LIN {X 0,Y 151.915,Z 503.399,A -85,B 0,C 180,E1 -24424.924,E2 -24424.924} C_VEL
LIN {X 0,Y 153.961,Z 512.067,A -85,B 0,C 180,E1 -24426.981,E2 -24426.981} C_VEL
LIN {X 0,Y 155.485,Z 521.164,A -85,B 0,C 180,E1 -24429.257,E2 -24429.257} C_VEL
LIN {X 0,Y 152.235,Z 533.845,A -85,B 0,C 180,E1 -24432.383,E2 -24432.383} C_VEL
LIN {X 0,Y 149.159,Z 545.494,A -85,B 0,C 180,E1 -24435.973,E2 -24435.973} C_VEL
LIN {X 0,Y 146.128,Z 556.818,A -85,B 0,C 180,E1 -24440.309,E2 -24440.309} C_VEL
LIN {X 0,Y 143.834,Z 566.337,A -85,B 0,C 180,E1 -24444.838,E2 -24444.838} C_VEL
LIN {X 0,Y 142.226,Z 574.336,A -85,B 0,C 180,E1 -24449.568,E2 -24449.568} C_VEL
LIN {X 0,Y 141.026,Z 581.744,A -85,B 0,C 180,E1 -24455.034,E2 -24455.034} C_VEL
LIN {X 0,Y 140.53,Z 587.875,A -85,B 0,C 180,E1 -24460.838,E2 -24460.838} C_VEL
LIN {X 0,Y 140.751,Z 591.758,A -85,B 0,C 180,E1 -24465.542,E2 -24465.542} C_VEL
LIN {X 0,Y 142.113,Z 595.406,A -85,B 0,C 180,E1 -24471.514,E2 -24471.514} C_VEL
LIN {X 0,Y 144.598,Z 597.709,A -85,B 0,C 180,E1 -24477.214,E2 -24477.214} C_VEL
LIN {X 0,Y 148.347,Z 598.825,A -85,B 0,C 180,E1 -24482.715,E2 -24482.715} C_VEL
LIN {X 0,Y 153.36,Z 598.771,A -85,B 0,C 180,E1 -24487.902,E2 -24487.902} C_VEL
LIN {X 0,Y 159.682,Z 597.562,A -85,B 0,C 180,E1 -24492.712,E2 -24492.712} C_VEL
LIN {X 0,Y 167.08,Z 595.209,A -85,B 0,C 180,E1 -24497.124,E2 -24497.124} C_VEL
LIN {X 0,Y 175.627,Z 591.631,A -85,B 0,C 180,E1 -24501.109,E2 -24501.109} C_VEL
LIN {X 0,Y 185.071,Z 586.803,A -85,B 0,C 180,E1 -24504.69,E2 -24504.69} C_VEL
LIN {X 0,Y 195.365,Z 580.517,A -85,B 0,C 180,E1 -24507.882,E2 -24507.882} C_VEL
LIN {X 0,Y 198.021,Z 578.731,A -85,B 0,C 180,E1 -24508.628,E2 -24508.628} C_VEL
LIN {X 0,Y 199.744,Z 577.522,A -85,B 0,C 180,E1 -24509.511,E2 -24509.511} C_VEL
LIN {X 0,Y 200.149,Z 577.047,A -85,B 0,C 180,E1 -24511.783,E2 -24511.783} C_VEL
LIN {X 0,Y 199.933,Z 577.424,A -85,B 0,C 180,E1 -24514.224,E2 -24514.224} C_VEL
LIN {X 0,Y 199.181,Z 578.642,A -85,B 0,C 180,E1 -24516.858,E2 -24516.858} C_VEL
LIN {X 0,Y 198.163,Z 580.069,A -85,B 0,C 180,E1 -24518.718,E2 -24518.718} C_VEL
LIN {X 0,Y 194.723,Z 583.259,A -85,B 0,C 180,E1 -24520.719,E2 -24520.719} C_VEL
LIN {X 0,Y 192.674,Z 584.987,A -85,B 0,C 180,E1 -24521.604,E2 -24521.604} C_VEL
LIN {X 0,Y 182.603,Z 591.982,A -85,B 0,C 180,E1 -24524.601,E2 -24524.601} C_VEL
LIN {X 0,Y 175.435,Z 596.39,A -85,B 0,C 180,E1 -24527.077,E2 -24527.077} C_VEL
LIN {X 0,Y 169.007,Z 600.188,A -85,B 0,C 180,E1 -24529.869,E2 -24529.869} C_VEL
LIN {X 0,Y 159.468,Z 605.111,A -85,B 0,C 180,E1 -24535.046,E2 -24535.046} C_VEL
LIN {X 0,Y 153.08,Z 607.936,A -85,B 0,C 180,E1 -24539.668,E2 -24539.668} C_VEL
LIN {X 0,Y 147.919,Z 609.705,A -85,B 0,C 180,E1 -24544.684,E2 -24544.684} C_VEL
LIN {X 0,Y 144.261,Z 610.461,A -85,B 0,C 180,E1 -24550.061,E2 -24550.061} C_VEL
LIN {X 0,Y 141.949,Z 610.176,A -85,B 0,C 180,E1 -24555.667,E2 -24555.667} C_VEL
LIN {X 0,Y 141.165,Z 608.842,A -85,B 0,C 180,E1 -24561.411,E2 -24561.411} C_VEL
LIN {X 0,Y 141.409,Z 606.295,A -85,B 0,C 180,E1 -24567.151,E2 -24567.151} C_VEL
LIN {X 0,Y 141.696,Z 604.494,A -85,B 0,C 180,E1 -24570,E2 -24570} C_VEL
LIN {X 0,Y 141.625,Z 600.931,A -85,B 0,C 180,E1 -24574.269,E2 -24574.269} C_VEL
LIN {X 0,Y 141.705,Z 596.358,A -85,B 0,C 180,E1 -24578.557,E2 -24578.557} C_VEL
LIN {X 0,Y 142.445,Z 589.643,A -85,B 0,C 180,E1 -24583.553,E2 -24583.553} C_VEL
LIN {X 0,Y 143.855,Z 581.253,A -85,B 0,C 180,E1 -24588.515,E2 -24588.515} C_VEL
LIN {X 0,Y 146.252,Z 571.401,A -85,B 0,C 180,E1 -24593.174,E2 -24593.174} C_VEL
LIN {X 0,Y 149.185,Z 560.252,A -85,B 0,C 180,E1 -24597.342,E2 -24597.342} C_VEL
LIN {X 0,Y 151.473,Z 551.924,A -85,B 0,C 180,E1 -24599.918,E2 -24599.918} C_VEL
LIN {X 0,Y 151.337,Z 542.468,A -85,B 0,C 180,E1 -24602.552,E2 -24602.552} C_VEL
LIN {X 0,Y 150.687,Z 529.752,A -85,B 0,C 180,E1 -24605.661,E2 -24605.661} C_VEL
LIN {X 0,Y 149.785,Z 516.716,A -85,B 0,C 180,E1 -24608.385,E2 -24608.385} C_VEL
LIN {X 0,Y 148.397,Z 501.688,A -85,B 0,C 180,E1 -24611.025,E2 -24611.025} C_VEL
LIN {X 0,Y 148.196,Z 499.899,A -85,B 0,C 180,E1 -24611.307,E2 -24611.307} C_VEL
LIN {X 0,Y 147.031,Z 496.512,A -85,B 0,C 180,E1 -24611.96,E2 -24611.96} C_VEL
LIN {X 0,Y 144.85,Z 493.641,A -85,B 0,C 180,E1 -24612.684,E2 -24612.684} C_VEL
LIN {X 0,Y 139.14,Z 487.285,A -85,B 0,C 180,E1 -24614.413,E2 -24614.413} C_VEL
LIN {X 0,Y 137.741,Z 483.867,A -85,B 0,C 180,E1 -24615.056,E2 -24615.056} C_VEL
LIN {X 0,Y 137.534,Z 482.616,A -85,B 0,C 180,E1 -24615.344,E2 -24615.344} C_VEL
LIN {X 0,Y 136.786,Z 479.643,A -85,B 0,C 180,E1 -24620.415,E2 -24620.415} C_VEL
LIN {X 0,Y 136.409,Z 477.116,A -85,B 0,C 180,E1 -24625.029,E2 -24625.029} C_VEL
LIN {X 0,Y 136.147,Z 477.149,A -85,B 0,C 180,E1 -24632.317,E2 -24632.317} C_VEL
LIN {X 0,Y 136.243,Z 477.139,A -85,B 0,C 180,E1 -24638.833,E2 -24638.833} C_VEL
LIN {X 0,Y 136.285,Z 477.129,A -85,B 0,C 180,E1 -24645.059,E2 -24645.059} C_VEL
LIN {X 0,Y 136.495,Z 477.107,A -85,B 0,C 180,E1 -24648.115,E2 -24648.115} C_VEL
LIN {X 0,Y 136.59,Z 477.092,A -85,B 0,C 180,E1 -24651.121,E2 -24651.121} C_VEL
LIN {X 0,Y 137.132,Z 477.026,A -85,B 0,C 180,E1 -24660.001,E2 -24660.001} C_VEL
LIN {X 0,Y 136.59,Z 477.092,A -85,B 0,C 180,E1 -24668.88,E2 -24668.88} C_VEL
LIN {X 0,Y 136.49,Z 477.103,A -85,B 0,C 180,E1 -24671.955,E2 -24671.955} C_VEL
LIN {X 0,Y 136.243,Z 477.136,A -85,B 0,C 180,E1 -24678.03,E2 -24678.03} C_VEL
LIN {X 0,Y 136.197,Z 477.142,A -85,B 0,C 180,E1 -24681.749,E2 -24681.749} C_VEL
LIN {X 0,Y 136.1,Z 477.151,A -85,B 0,C 180,E1 -24688.617,E2 -24688.617} C_VEL
LIN {X 0,Y 136.079,Z 477.157,A -85,B 0,C 180,E1 -24694.62,E2 -24694.62} C_VEL
LIN {X 0,Y 136.051,Z 477.16,A -85,B 0,C 180,E1 -24699.209,E2 -24699.209} C_VEL
LIN {X 0,Y 136.004,Z 477.168,A -85,B 0,C 180,E1 -24703.661,E2 -24703.661} C_VEL
LIN {X 0,Y 136.036,Z 477.162,A -85,B 0,C 180,E1 -24707.809,E2 -24707.809} C_VEL
LIN {X 0,Y 136.058,Z 477.162,A -85,B 0,C 180,E1 -24711.695,E2 -24711.695} C_VEL
LIN {X 0,Y 136.092,Z 477.152,A -85,B 0,C 180,E1 -24715.718,E2 -24715.718} C_VEL
LIN {X 0,Y 136.149,Z 477.145,A -85,B 0,C 180,E1 -24722.317,E2 -24722.317} C_VEL
LIN {X 0,Y 136.246,Z 477.138,A -85,B 0,C 180,E1 -24728.834,E2 -24728.834} C_VEL
LIN {X 0,Y 136.271,Z 477.134,A -85,B 0,C 180,E1 -24735.057,E2 -24735.057} C_VEL
LIN {X 0,Y 136.434,Z 477.113,A -85,B 0,C 180,E1 -24738.165,E2 -24738.165} C_VEL
LIN {X 0,Y 136.552,Z 477.094,A -85,B 0,C 180,E1 -24741.118,E2 -24741.118} C_VEL
LIN {X 0,Y 137.136,Z 477.021,A -85,B 0,C 180,E1 -24750,E2 -24750} C_VEL
LIN {X 0,Y 136.556,Z 477.091,A -85,B 0,C 180,E1 -24758.882,E2 -24758.882} C_VEL
LIN {X 0,Y 136.443,Z 477.113,A -85,B 0,C 180,E1 -24761.89,E2 -24761.89} C_VEL
LIN {X 0,Y 136.249,Z 477.134,A -85,B 0,C 180,E1 -24768.028,E2 -24768.028} C_VEL
LIN {X 0,Y 136.201,Z 477.144,A -85,B 0,C 180,E1 -24771.749,E2 -24771.749} C_VEL
LIN {X 0,Y 136.166,Z 477.215,A -85,B 0,C 180,E1 -24778.003,E2 -24778.003} C_VEL
LIN {X 0,Y 137.968,Z 482.338,A -85,B 0,C 180,E1 -24779.083,E2 -24779.083} C_VEL
LIN {X 0,Y 142.002,Z 494.173,A -85,B 0,C 180,E1 -24781.725,E2 -24781.725} C_VEL
LIN {X 0,Y 145.517,Z 506.485,A -85,B 0,C 180,E1 -24784.659,E2 -24784.659} C_VEL
LIN {X 0,Y 147.515,Z 515.552,A -85,B 0,C 180,E1 -24786.976,E2 -24786.976} C_VEL
LIN {X 0,Y 148.445,Z 520.908,A -85,B 0,C 180,E1 -24788.417,E2 -24788.417} C_VEL
LIN {X 0,Y 147.335,Z 526.449,A -85,B 0,C 180,E1 -24789.772,E2 -24789.772} C_VEL
LIN {X 0,Y 143.953,Z 538.976,A -85,B 0,C 180,E1 -24793.272,E2 -24793.272} C_VEL
LIN {X 0,Y 140.81,Z 550.38,A -85,B 0,C 180,E1 -24797.298,E2 -24797.298} C_VEL
LIN {X 0,Y 138.22,Z 559.95,A -85,B 0,C 180,E1 -24801.473,E2 -24801.473} C_VEL
LIN {X 0,Y 136.13,Z 569.001,A -85,B 0,C 180,E1 -24806.319,E2 -24806.319} C_VEL
LIN {X 0,Y 134.673,Z 576.356,A -85,B 0,C 180,E1 -24811.136,E2 -24811.136} C_VEL
LIN {X 0,Y 133.697,Z 583.307,A -85,B 0,C 180,E1 -24816.78,E2 -24816.78} C_VEL
LIN {X 0,Y 133.467,Z 588.029,A -85,B 0,C 180,E1 -24821.582,E2 -24821.582} C_VEL
LIN {X 0,Y 134.029,Z 592.858,A -85,B 0,C 180,E1 -24827.892,E2 -24827.892} C_VEL
LIN {X 0,Y 135.854,Z 596.28,A -85,B 0,C 180,E1 -24834.061,E2 -24834.061} C_VEL
LIN {X 0,Y 138.982,Z 598.438,A -85,B 0,C 180,E1 -24839.999,E2 -24839.999} C_VEL
LIN {X 0,Y 143.394,Z 599.427,A -85,B 0,C 180,E1 -24845.625,E2 -24845.625} C_VEL
LIN {X 0,Y 149.209,Z 599.265,A -85,B 0,C 180,E1 -24850.859,E2 -24850.859} C_VEL
LIN {X 0,Y 156.236,Z 597.981,A -85,B 0,C 180,E1 -24855.658,E2 -24855.658} C_VEL
LIN {X 0,Y 164.656,Z 595.448,A -85,B 0,C 180,E1 -24860.115,E2 -24860.115} C_VEL
LIN {X 0,Y 173.636,Z 591.918,A -85,B 0,C 180,E1 -24863.875,E2 -24863.875} C_VEL
LIN {X 0,Y 183.769,Z 586.966,A -85,B 0,C 180,E1 -24867.317,E2 -24867.317} C_VEL
LIN {X 0,Y 191.889,Z 582.364,A -85,B 0,C 180,E1 -24869.633,E2 -24869.633} C_VEL
LIN {X 0,Y 193.883,Z 581.13,A -85,B 0,C 180,E1 -24870.496,E2 -24870.496} C_VEL
LIN {X 0,Y 194.153,Z 581.028,A -85,B 0,C 180,E1 -24872.886,E2 -24872.886} C_VEL
LIN {X 0,Y 193.576,Z 581.831,A -85,B 0,C 180,E1 -24875.513,E2 -24875.513} C_VEL
LIN {X 0,Y 193.043,Z 582.549,A -85,B 0,C 180,E1 -24876.781,E2 -24876.781} C_VEL
LIN {X 0,Y 191.011,Z 584.458,A -85,B 0,C 180,E1 -24878.718,E2 -24878.718} C_VEL
LIN {X 0,Y 188.142,Z 586.678,A -85,B 0,C 180,E1 -24880.025,E2 -24880.025} C_VEL
LIN {X 0,Y 175.247,Z 594.662,A -85,B 0,C 180,E1 -24883.793,E2 -24883.793} C_VEL
LIN {X 0,Y 170.358,Z 597.377,A -85,B 0,C 180,E1 -24885.468,E2 -24885.468} C_VEL
LIN {X 0,Y 163.66,Z 600.823,A -85,B 0,C 180,E1 -24888.272,E2 -24888.272} C_VEL
LIN {X 0,Y 153.705,Z 605.368,A -85,B 0,C 180,E1 -24893.53,E2 -24893.53} C_VEL
LIN {X 0,Y 146.976,Z 607.866,A -85,B 0,C 180,E1 -24898.266,E2 -24898.266} C_VEL
LIN {X 0,Y 141.496,Z 609.39,A -85,B 0,C 180,E1 -24903.448,E2 -24903.448} C_VEL
LIN {X 0,Y 137.583,Z 609.931,A -85,B 0,C 180,E1 -24909.049,E2 -24909.049} C_VEL
LIN {X 0,Y 135.057,Z 609.412,A -85,B 0,C 180,E1 -24914.919,E2 -24914.919} C_VEL
LIN {X 0,Y 134.187,Z 607.83,A -85,B 0,C 180,E1 -24920.96,E2 -24920.96} C_VEL
LIN {X 0,Y 134.429,Z 605.091,A -85,B 0,C 180,E1 -24927.003,E2 -24927.003} C_VEL
LIN {X 0,Y 134.703,Z 603.171,A -85,B 0,C 180,E1 -24930,E2 -24930} C_VEL
LIN {X 0,Y 134.639,Z 599.417,A -85,B 0,C 180,E1 -24934.491,E2 -24934.491} C_VEL
LIN {X 0,Y 134.737,Z 594.629,A -85,B 0,C 180,E1 -24939.003,E2 -24939.003} C_VEL
LIN {X 0,Y 135.531,Z 587.676,A -85,B 0,C 180,E1 -24944.259,E2 -24944.259} C_VEL
LIN {X 0,Y 137.169,Z 578.999,A -85,B 0,C 180,E1 -24949.453,E2 -24949.453} C_VEL
LIN {X 0,Y 139.771,Z 568.81,A -85,B 0,C 180,E1 -24954.272,E2 -24954.272} C_VEL
LIN {X 0,Y 142.942,Z 557.155,A -85,B 0,C 180,E1 -24958.644,E2 -24958.644} C_VEL
LIN {X 0,Y 144.449,Z 551.841,A -85,B 0,C 180,E1 -24960.316,E2 -24960.316} C_VEL
LIN {X 0,Y 144.245,Z 540.81,A -85,B 0,C 180,E1 -24963.545,E2 -24963.545} C_VEL
LIN {X 0,Y 143.651,Z 528.627,A -85,B 0,C 180,E1 -24966.643,E2 -24966.643} C_VEL
LIN {X 0,Y 142.67,Z 513.871,A -85,B 0,C 180,E1 -24969.82,E2 -24969.82} C_VEL
LIN {X 0,Y 141.296,Z 498.785,A -85,B 0,C 180,E1 -24972.544,E2 -24972.544} C_VEL
LIN {X 0,Y 139.832,Z 490.806,A -85,B 0,C 180,E1 -24973.87,E2 -24973.87} C_VEL
LIN {X 0,Y 137.741,Z 483.867,A -85,B 0,C 180,E1 -24975.056,E2 -24975.056} C_VEL
LIN {X 0,Y 137.192,Z 482.692,A -85,B 0,C 180,E1 -24975.528,E2 -24975.528} C_VEL
LIN {X 0,Y 132.35,Z 480.042,A -85,B 0,C 180,E1 -24980.631,E2 -24980.631} C_VEL
LIN {X 0,Y 129.515,Z 478.302,A -85,B 0,C 180,E1 -24985.878,E2 -24985.878} C_VEL
LIN {X 0,Y 129.14,Z 478.017,A -85,B 0,C 180,E1 -24987.864,E2 -24987.864} C_VEL
LIN {X 0,Y 129.03,Z 478.027,A -85,B 0,C 180,E1 -24994.168,E2 -24994.168} C_VEL
LIN {X 0,Y 129.106,Z 478.026,A -85,B 0,C 180,E1 -24997.728,E2 -24997.728} C_VEL
LIN {X 0,Y 129.161,Z 478.021,A -85,B 0,C 180,E1 -25000.946,E2 -25000.946} C_VEL
LIN {X 0,Y 129.415,Z 477.988,A -85,B 0,C 180,E1 -25007.821,E2 -25007.821} C_VEL
LIN {X 0,Y 129.515,Z 477.975,A -85,B 0,C 180,E1 -25010.632,E2 -25010.632} C_VEL
LIN {X 0,Y 130.087,Z 477.904,A -85,B 0,C 180,E1 -25020.001,E2 -25020.001} C_VEL
LIN {X 0,Y 129.516,Z 477.972,A -85,B 0,C 180,E1 -25029.37,E2 -25029.37} C_VEL
LIN {X 0,Y 129.392,Z 477.989,A -85,B 0,C 180,E1 -25032.549,E2 -25032.549} C_VEL
LIN {X 0,Y 129.153,Z 478.014,A -85,B 0,C 180,E1 -25039.057,E2 -25039.057} C_VEL
LIN {X 0,Y 129.108,Z 478.027,A -85,B 0,C 180,E1 -25042.399,E2 -25042.399} C_VEL
LIN {X 0,Y 129.035,Z 478.031,A -85,B 0,C 180,E1 -25049.374,E2 -25049.374} C_VEL
LIN {X 0,Y 128.992,Z 478.039,A -85,B 0,C 180,E1 -25055.19,E2 -25055.19} C_VEL
LIN {X 0,Y 128.952,Z 478.047,A -85,B 0,C 180,E1 -25060.846,E2 -25060.846} C_VEL
LIN {X 0,Y 128.926,Z 478.045,A -85,B 0,C 180,E1 -25065.127,E2 -25065.127} C_VEL
LIN {X 0,Y 128.96,Z 478.046,A -85,B 0,C 180,E1 -25069.728,E2 -25069.728} C_VEL
LIN {X 0,Y 128.993,Z 478.034,A -85,B 0,C 180,E1 -25074.812,E2 -25074.812} C_VEL
LIN {X 0,Y 129.053,Z 478.033,A -85,B 0,C 180,E1 -25080.652,E2 -25080.652} C_VEL
LIN {X 0,Y 129.11,Z 478.029,A -85,B 0,C 180,E1 -25087.728,E2 -25087.728} C_VEL
LIN {X 0,Y 129.156,Z 478.018,A -85,B 0,C 180,E1 -25090.945,E2 -25090.945} C_VEL
LIN {X 0,Y 129.392,Z 477.991,A -85,B 0,C 180,E1 -25097.876,E2 -25097.876} C_VEL
LIN {X 0,Y 129.475,Z 477.975,A -85,B 0,C 180,E1 -25100.628,E2 -25100.628} C_VEL
LIN {X 0,Y 130.091,Z 477.899,A -85,B 0,C 180,E1 -25110,E2 -25110} C_VEL
LIN {X 0,Y 129.481,Z 477.971,A -85,B 0,C 180,E1 -25119.371,E2 -25119.371} C_VEL
LIN {X 0,Y 129.347,Z 477.997,A -85,B 0,C 180,E1 -25122.552,E2 -25122.552} C_VEL
LIN {X 0,Y 129.159,Z 478.02,A -85,B 0,C 180,E1 -25129.055,E2 -25129.055} C_VEL
LIN {X 0,Y 129.111,Z 478.026,A -85,B 0,C 180,E1 -25132.398,E2 -25132.398} C_VEL
LIN {X 0,Y 129.061,Z 478.12,A -85,B 0,C 180,E1 -25136.695,E2 -25136.695} C_VEL
LIN {X 0,Y 134.061,Z 491.907,A -85,B 0,C 180,E1 -25139.983,E2 -25139.983} C_VEL
LIN {X 0,Y 138.043,Z 505.591,A -85,B 0,C 180,E1 -25143.399,E2 -25143.399} C_VEL
LIN {X 0,Y 140.382,Z 515.395,A -85,B 0,C 180,E1 -25146.033,E2 -25146.033} C_VEL
LIN {X 0,Y 141.506,Z 521.96,A -85,B 0,C 180,E1 -25147.87,E2 -25147.87} C_VEL
LIN {X 0,Y 138.858,Z 532.205,A -85,B 0,C 180,E1 -25150.606,E2 -25150.606} C_VEL
LIN {X 0,Y 135.498,Z 544.203,A -85,B 0,C 180,E1 -25154.504,E2 -25154.504} C_VEL
LIN {X 0,Y 132.618,Z 554.392,A -85,B 0,C 180,E1 -25158.61,E2 -25158.61} C_VEL
LIN {X 0,Y 130.029,Z 564.246,A -85,B 0,C 180,E1 -25163.519,E2 -25163.519} C_VEL
LIN {X 0,Y 128.262,Z 572.581,A -85,B 0,C 180,E1 -25168.63,E2 -25168.63} C_VEL
LIN {X 0,Y 127.06,Z 579.338,A -85,B 0,C 180,E1 -25173.736,E2 -25173.736} C_VEL
LIN {X 0,Y 126.47,Z 584.855,A -85,B 0,C 180,E1 -25178.825,E2 -25178.825} C_VEL
LIN {X 0,Y 126.468,Z 589.328,A -85,B 0,C 180,E1 -25183.867,E2 -25183.867} C_VEL
LIN {X 0,Y 127.495,Z 593.911,A -85,B 0,C 180,E1 -25190.481,E2 -25190.481} C_VEL
LIN {X 0,Y 129.891,Z 597.149,A -85,B 0,C 180,E1 -25196.898,E2 -25196.898} C_VEL
LIN {X 0,Y 133.714,Z 599.163,A -85,B 0,C 180,E1 -25203.012,E2 -25203.012} C_VEL
LIN {X 0,Y 138.879,Z 600.033,A -85,B 0,C 180,E1 -25208.732,E2 -25208.732} C_VEL
LIN {X 0,Y 145.476,Z 599.777,A -85,B 0,C 180,E1 -25213.978,E2 -25213.978} C_VEL
LIN {X 0,Y 153.285,Z 598.402,A -85,B 0,C 180,E1 -25218.72,E2 -25218.72} C_VEL
LIN {X 0,Y 162.236,Z 595.908,A -85,B 0,C 180,E1 -25222.946,E2 -25222.946} C_VEL
LIN {X 0,Y 174.014,Z 591.404,A -85,B 0,C 180,E1 -25227.314,E2 -25227.314} C_VEL
LIN {X 0,Y 185.753,Z 585.748,A -85,B 0,C 180,E1 -25230.715,E2 -25230.715} C_VEL
LIN {X 0,Y 187.831,Z 584.649,A -85,B 0,C 180,E1 -25231.589,E2 -25231.589} C_VEL
LIN {X 0,Y 187.628,Z 585.102,A -85,B 0,C 180,E1 -25234.509,E2 -25234.509} C_VEL
LIN {X 0,Y 185.715,Z 586.956,A -85,B 0,C 180,E1 -25237.374,E2 -25237.374} C_VEL
LIN {X 0,Y 183.734,Z 588.294,A -85,B 0,C 180,E1 -25238.36,E2 -25238.36} C_VEL
LIN {X 0,Y 173.087,Z 594.39,A -85,B 0,C 180,E1 -25241.309,E2 -25241.309} C_VEL
LIN {X 0,Y 165.424,Z 598.216,A -85,B 0,C 180,E1 -25243.761,E2 -25243.761} C_VEL
LIN {X 0,Y 156.267,Z 602.386,A -85,B 0,C 180,E1 -25247.577,E2 -25247.577} C_VEL
LIN {X 0,Y 148.063,Z 605.57,A -85,B 0,C 180,E1 -25251.899,E2 -25251.899} C_VEL
LIN {X 0,Y 140.958,Z 607.803,A -85,B 0,C 180,E1 -25256.74,E2 -25256.74} C_VEL
LIN {X 0,Y 134.935,Z 609.055,A -85,B 0,C 180,E1 -25262.304,E2 -25262.304} C_VEL
LIN {X 0,Y 130.955,Z 609.281,A -85,B 0,C 180,E1 -25267.935,E2 -25267.935} C_VEL
LIN {X 0,Y 128.205,Z 608.53,A -85,B 0,C 180,E1 -25274.092,E2 -25274.092} C_VEL
LIN {X 0,Y 127.223,Z 606.785,A -85,B 0,C 180,E1 -25280.461,E2 -25280.461} C_VEL
LIN {X 0,Y 127.444,Z 603.819,A -85,B 0,C 180,E1 -25286.839,E2 -25286.839} C_VEL
LIN {X 0,Y 127.71,Z 601.799,A -85,B 0,C 180,E1 -25290,E2 -25290} C_VEL
LIN {X 0,Y 127.651,Z 597.833,A -85,B 0,C 180,E1 -25294.737,E2 -25294.737} C_VEL
LIN {X 0,Y 127.79,Z 592.798,A -85,B 0,C 180,E1 -25299.496,E2 -25299.496} C_VEL
LIN {X 0,Y 128.712,Z 585.516,A -85,B 0,C 180,E1 -25305.032,E2 -25305.032} C_VEL
LIN {X 0,Y 130.514,Z 576.494,A -85,B 0,C 180,E1 -25310.488,E2 -25310.488} C_VEL
LIN {X 0,Y 133.014,Z 567.2,A -85,B 0,C 180,E1 -25315.004,E2 -25315.004} C_VEL
LIN {X 0,Y 136.167,Z 556.028,A -85,B 0,C 180,E1 -25319.361,E2 -25319.361} C_VEL
LIN {X 0,Y 137.393,Z 551.736,A -85,B 0,C 180,E1 -25320.765,E2 -25320.765} C_VEL
LIN {X 0,Y 137.277,Z 541.887,A -85,B 0,C 180,E1 -25323.831,E2 -25323.831} C_VEL
LIN {X 0,Y 136.732,Z 529.428,A -85,B 0,C 180,E1 -25327.206,E2 -25327.206} C_VEL
LIN {X 0,Y 135.861,Z 514.85,A -85,B 0,C 180,E1 -25330.558,E2 -25330.558} C_VEL
LIN {X 0,Y 134.605,Z 499.779,A -85,B 0,C 180,E1 -25333.442,E2 -25333.442} C_VEL
LIN {X 0,Y 133.074,Z 491.845,A -85,B 0,C 180,E1 -25334.891,E2 -25334.891} C_VEL
LIN {X 0,Y 130.204,Z 482.203,A -85,B 0,C 180,E1 -25336.78,E2 -25336.78} C_VEL
LIN {X 0,Y 129.404,Z 477.991,A -85,B 0,C 180,E1 -25344.552,E2 -25344.552} C_VEL
LIN {X 0,Y 129.14,Z 478.017,A -85,B 0,C 180,E1 -25347.864,E2 -25347.864} C_VEL
LIN {X 0,Y 128.327,Z 478.127,A -85,B 0,C 180,E1 -25350.467,E2 -25350.467} C_VEL
LIN {X 0,Y 126.69,Z 478.323,A -85,B 0,C 180,E1 -25353.036,E2 -25353.036} C_VEL
LIN {X 0,Y 122.283,Z 478.877,A -85,B 0,C 180,E1 -25360.148,E2 -25360.148} C_VEL
LIN {X 0,Y 122.042,Z 478.897,A -85,B 0,C 180,E1 -25362.027,E2 -25362.027} C_VEL
LIN {X 0,Y 122.362,Z 478.867,A -85,B 0,C 180,E1 -25367.527,E2 -25367.527} C_VEL
LIN {X 0,Y 122.445,Z 478.857,A -85,B 0,C 180,E1 -25370.085,E2 -25370.085} C_VEL
LIN {X 0,Y 122.605,Z 478.838,A -85,B 0,C 180,E1 -25376.715,E2 -25376.715} C_VEL
LIN {X 0,Y 123.041,Z 478.781,A -85,B 0,C 180,E1 -25380.001,E2 -25380.001} C_VEL
LIN {X 0,Y 122.419,Z 478.857,A -85,B 0,C 180,E1 -25387.113,E2 -25387.113} C_VEL
LIN {X 0,Y 122.362,Z 478.864,A -85,B 0,C 180,E1 -25392.474,E2 -25392.474} C_VEL
LIN {X 0,Y 122.045,Z 478.901,A -85,B 0,C 180,E1 -25400.214,E2 -25400.214} C_VEL
LIN {X 0,Y 121.983,Z 478.915,A -85,B 0,C 180,E1 -25403.786,E2 -25403.786} C_VEL
LIN {X 0,Y 121.942,Z 478.917,A -85,B 0,C 180,E1 -25410.175,E2 -25410.175} C_VEL
LIN {X 0,Y 121.912,Z 478.917,A -85,B 0,C 180,E1 -25416.19,E2 -25416.19} C_VEL
LIN {X 0,Y 121.886,Z 478.927,A -85,B 0,C 180,E1 -25421.447,E2 -25421.447} C_VEL
LIN {X 0,Y 121.887,Z 478.926,A -85,B 0,C 180,E1 -25428.555,E2 -25428.555} C_VEL
LIN {X 0,Y 121.946,Z 478.912,A -85,B 0,C 180,E1 -25434.809,E2 -25434.809} C_VEL
LIN {X 0,Y 121.944,Z 478.92,A -85,B 0,C 180,E1 -25439.827,E2 -25439.827} C_VEL
LIN {X 0,Y 121.986,Z 478.914,A -85,B 0,C 180,E1 -25446.216,E2 -25446.216} C_VEL
LIN {X 0,Y 122.048,Z 478.905,A -85,B 0,C 180,E1 -25449.788,E2 -25449.788} C_VEL
LIN {X 0,Y 122.242,Z 478.882,A -85,B 0,C 180,E1 -25456.705,E2 -25456.705} C_VEL
LIN {X 0,Y 122.411,Z 478.856,A -85,B 0,C 180,E1 -25460.082,E2 -25460.082} C_VEL
LIN {X 0,Y 122.598,Z 478.838,A -85,B 0,C 180,E1 -25466.714,E2 -25466.714} C_VEL
LIN {X 0,Y 123.044,Z 478.776,A -85,B 0,C 180,E1 -25470,E2 -25470} C_VEL
LIN {X 0,Y 122.431,Z 478.857,A -85,B 0,C 180,E1 -25476.592,E2 -25476.592} C_VEL
LIN {X 0,Y 122.32,Z 478.872,A -85,B 0,C 180,E1 -25482.376,E2 -25482.376} C_VEL
LIN {X 0,Y 122.114,Z 478.898,A -85,B 0,C 180,E1 -25486.724,E2 -25486.724} C_VEL
LIN {X 0,Y 122.025,Z 478.908,A -85,B 0,C 180,E1 -25492.849,E2 -25492.849} C_VEL
LIN {X 0,Y 122.006,Z 479.113,A -85,B 0,C 180,E1 -25495.367,E2 -25495.367} C_VEL
LIN {X 0,Y 127.149,Z 493.141,A -85,B 0,C 180,E1 -25498.923,E2 -25498.923} C_VEL
LIN {X 0,Y 130.636,Z 504.946,A -85,B 0,C 180,E1 -25502.09,E2 -25502.09} C_VEL
LIN {X 0,Y 133.473,Z 516.49,A -85,B 0,C 180,E1 -25505.394,E2 -25505.394} C_VEL
LIN {X 0,Y 134.459,Z 523.125,A -85,B 0,C 180,E1 -25507.357,E2 -25507.357} C_VEL
LIN {X 0,Y 131.243,Z 534.715,A -85,B 0,C 180,E1 -25510.665,E2 -25510.665} C_VEL
LIN {X 0,Y 127.758,Z 546.719,A -85,B 0,C 180,E1 -25514.953,E2 -25514.953} C_VEL
LIN {X 0,Y 124.717,Z 557.165,A -85,B 0,C 180,E1 -25519.605,E2 -25519.605} C_VEL
LIN {X 0,Y 122.334,Z 566.717,A -85,B 0,C 180,E1 -25524.935,E2 -25524.935} C_VEL
LIN {X 0,Y 120.78,Z 574.066,A -85,B 0,C 180,E1 -25529.949,E2 -25529.949} C_VEL
LIN {X 0,Y 119.715,Z 581.032,A -85,B 0,C 180,E1 -25535.735,E2 -25535.735} C_VEL
LIN {X 0,Y 119.307,Z 586.794,A -85,B 0,C 180,E1 -25541.671,E2 -25541.671} C_VEL
LIN {X 0,Y 119.869,Z 591.758,A -85,B 0,C 180,E1 -25548.158,E2 -25548.158} C_VEL
LIN {X 0,Y 121.23,Z 594.933,A -85,B 0,C 180,E1 -25553.341,E2 -25553.341} C_VEL
LIN {X 0,Y 124.269,Z 597.991,A -85,B 0,C 180,E1 -25559.999,E2 -25559.999} C_VEL
LIN {X 0,Y 128.83,Z 599.882,A -85,B 0,C 180,E1 -25566.263,E2 -25566.263} C_VEL
LIN {X 0,Y 134.849,Z 600.644,A -85,B 0,C 180,E1 -25572.032,E2 -25572.032} C_VEL
LIN {X 0,Y 142.23,Z 600.303,A -85,B 0,C 180,E1 -25577.246,E2 -25577.246} C_VEL
LIN {X 0,Y 152.109,Z 598.599,A -85,B 0,C 180,E1 -25582.473,E2 -25582.473} C_VEL
LIN {X 0,Y 160.543,Z 596.31,A -85,B 0,C 180,E1 -25585.961,E2 -25585.961} C_VEL
LIN {X 0,Y 171.119,Z 592.579,A -85,B 0,C 180,E1 -25589.528,E2 -25589.528} C_VEL
LIN {X 0,Y 179.638,Z 588.945,A -85,B 0,C 180,E1 -25591.881,E2 -25591.881} C_VEL
LIN {X 0,Y 181.471,Z 588.137,A -85,B 0,C 180,E1 -25592.832,E2 -25592.832} C_VEL
LIN {X 0,Y 180.62,Z 588.957,A -85,B 0,C 180,E1 -25595.204,E2 -25595.204} C_VEL
LIN {X 0,Y 180.242,Z 589.302,A -85,B 0,C 180,E1 -25595.794,E2 -25595.794} C_VEL
LIN {X 0,Y 178.984,Z 590.172,A -85,B 0,C 180,E1 -25596.768,E2 -25596.768} C_VEL
LIN {X 0,Y 165.846,Z 596.744,A -85,B 0,C 180,E1 -25600.291,E2 -25600.291} C_VEL
LIN {X 0,Y 155.708,Z 601.084,A -85,B 0,C 180,E1 -25603.767,E2 -25603.767} C_VEL
LIN {X 0,Y 146.681,Z 604.415,A -85,B 0,C 180,E1 -25607.873,E2 -25607.873} C_VEL
LIN {X 0,Y 138.664,Z 606.769,A -85,B 0,C 180,E1 -25612.541,E2 -25612.541} C_VEL
LIN {X 0,Y 131.813,Z 608.211,A -85,B 0,C 180,E1 -25617.78,E2 -25617.78} C_VEL
LIN {X 0,Y 126.448,Z 608.719,A -85,B 0,C 180,E1 -25623.6,E2 -25623.6} C_VEL
LIN {X 0,Y 122.644,Z 608.235,A -85,B 0,C 180,E1 -25629.89,E2 -25629.89} C_VEL
LIN {X 0,Y 120.664,Z 606.738,A -85,B 0,C 180,E1 -25636.528,E2 -25636.528} C_VEL
LIN {X 0,Y 120.274,Z 604.143,A -85,B 0,C 180,E1 -25643.392,E2 -25643.392} C_VEL
LIN {X 0,Y 120.612,Z 601.434,A -85,B 0,C 180,E1 -25648.33,E2 -25648.33} C_VEL
LIN {X 0,Y 120.698,Z 599.033,A -85,B 0,C 180,E1 -25651.668,E2 -25651.668} C_VEL
LIN {X 0,Y 120.687,Z 594.493,A -85,B 0,C 180,E1 -25656.688,E2 -25656.688} C_VEL
LIN {X 0,Y 121.196,Z 587.86,A -85,B 0,C 180,E1 -25662.56,E2 -25662.56} C_VEL
LIN {X 0,Y 122.573,Z 579.515,A -85,B 0,C 180,E1 -25668.382,E2 -25668.382} C_VEL
LIN {X 0,Y 125.185,Z 569.28,A -85,B 0,C 180,E1 -25674.017,E2 -25674.017} C_VEL
LIN {X 0,Y 128.235,Z 558.41,A -85,B 0,C 180,E1 -25678.731,E2 -25678.731} C_VEL
LIN {X 0,Y 130.395,Z 551.416,A -85,B 0,C 180,E1 -25681.249,E2 -25681.249} C_VEL
LIN {X 0,Y 130.15,Z 539.899,A -85,B 0,C 180,E1 -25685.008,E2 -25685.008} C_VEL
LIN {X 0,Y 129.655,Z 527.238,A -85,B 0,C 180,E1 -25688.561,E2 -25688.561} C_VEL
LIN {X 0,Y 128.899,Z 513.204,A -85,B 0,C 180,E1 -25691.895,E2 -25691.895} C_VEL
LIN {X 0,Y 127.799,Z 499.673,A -85,B 0,C 180,E1 -25694.646,E2 -25694.646} C_VEL
LIN {X 0,Y 126.009,Z 491.785,A -85,B 0,C 180,E1 -25696.26,E2 -25696.26} C_VEL
LIN {X 0,Y 122.908,Z 481.801,A -85,B 0,C 180,E1 -25698.323,E2 -25698.323} C_VEL
LIN {X 0,Y 122.368,Z 478.868,A -85,B 0,C 180,E1 -25704.223,E2 -25704.223} C_VEL
LIN {X 0,Y 122.036,Z 478.91,A -85,B 0,C 180,E1 -25709.749,E2 -25709.749} C_VEL
LIN {X 0,Y 122.022,Z 478.907,A -85,B 0,C 180,E1 -25717.149,E2 -25717.149} C_VEL
LIN {X 0,Y 122.042,Z 478.897,A -85,B 0,C 180,E1 -25722.027,E2 -25722.027} C_VEL
LIN {X 0,Y 121.46,Z 478.975,A -85,B 0,C 180,E1 -25724.785,E2 -25724.785} C_VEL
LIN {X 0,Y 119.95,Z 479.171,A -85,B 0,C 180,E1 -25727.513,E2 -25727.513} C_VEL
LIN {X 0,Y 115.728,Z 479.699,A -85,B 0,C 180,E1 -25735.075,E2 -25735.075} C_VEL
LIN {X 0,Y 115.575,Z 479.709,A -85,B 0,C 180,E1 -25737.068,E2 -25737.068} C_VEL
LIN {X 0,Y 115.993,Z 479.659,A -85,B 0,C 180,E1 -25740.001,E2 -25740.001} C_VEL
LIN {X 0,Y 115.388,Z 479.736,A -85,B 0,C 180,E1 -25747.001,E2 -25747.001} C_VEL
LIN {X 0,Y 115.283,Z 479.747,A -85,B 0,C 180,E1 -25752.738,E2 -25752.738} C_VEL
LIN {X 0,Y 115.012,Z 479.78,A -85,B 0,C 180,E1 -25757.791,E2 -25757.791} C_VEL
LIN {X 0,Y 114.946,Z 479.791,A -85,B 0,C 180,E1 -25763.493,E2 -25763.493} C_VEL
LIN {X 0,Y 114.869,Z 479.8,A -85,B 0,C 180,E1 -25771.069,E2 -25771.069} C_VEL
LIN {X 0,Y 114.802,Z 479.802,A -85,B 0,C 180,E1 -25777.749,E2 -25777.749} C_VEL
LIN {X 0,Y 114.797,Z 479.809,A -85,B 0,C 180,E1 -25782.723,E2 -25782.723} C_VEL
LIN {X 0,Y 114.806,Z 479.805,A -85,B 0,C 180,E1 -25787.672,E2 -25787.672} C_VEL
LIN {X 0,Y 114.814,Z 479.805,A -85,B 0,C 180,E1 -25792.728,E2 -25792.728} C_VEL
LIN {X 0,Y 114.87,Z 479.801,A -85,B 0,C 180,E1 -25798.933,E2 -25798.933} C_VEL
LIN {X 0,Y 114.949,Z 479.79,A -85,B 0,C 180,E1 -25806.508,E2 -25806.508} C_VEL
LIN {X 0,Y 115.014,Z 479.776,A -85,B 0,C 180,E1 -25812.21,E2 -25812.21} C_VEL
LIN {X 0,Y 115.251,Z 479.754,A -85,B 0,C 180,E1 -25817.341,E2 -25817.341} C_VEL
LIN {X 0,Y 115.366,Z 479.736,A -85,B 0,C 180,E1 -25823.002,E2 -25823.002} C_VEL
LIN {X 0,Y 115.996,Z 479.654,A -85,B 0,C 180,E1 -25830,E2 -25830} C_VEL
LIN {X 0,Y 115.371,Z 479.735,A -85,B 0,C 180,E1 -25836.998,E2 -25836.998} C_VEL
LIN {X 0,Y 115.255,Z 479.753,A -85,B 0,C 180,E1 -25842.667,E2 -25842.667} C_VEL
LIN {X 0,Y 115.016,Z 479.779,A -85,B 0,C 180,E1 -25847.789,E2 -25847.789} C_VEL
LIN {X 0,Y 114.952,Z 479.8,A -85,B 0,C 180,E1 -25853.81,E2 -25853.81} C_VEL
LIN {X 0,Y 120.303,Z 494.401,A -85,B 0,C 180,E1 -25857.862,E2 -25857.862} C_VEL
LIN {X 0,Y 123.746,Z 506.077,A -85,B 0,C 180,E1 -25861.193,E2 -25861.193} C_VEL
LIN {X 0,Y 126.601,Z 517.555,A -85,B 0,C 180,E1 -25864.68,E2 -25864.68} C_VEL
LIN {X 0,Y 127.455,Z 524.069,A -85,B 0,C 180,E1 -25866.735,E2 -25866.735} C_VEL
LIN {X 0,Y 123.761,Z 536.611,A -85,B 0,C 180,E1 -25870.577,E2 -25870.577} C_VEL
LIN {X 0,Y 120.045,Z 548.852,A -85,B 0,C 180,E1 -25875.368,E2 -25875.368} C_VEL
LIN {X 0,Y 117.015,Z 559.264,A -85,B 0,C 180,E1 -25880.498,E2 -25880.498} C_VEL
LIN {X 0,Y 114.651,Z 569.032,A -85,B 0,C 180,E1 -25886.516,E2 -25886.516} C_VEL
LIN {X 0,Y 113.185,Z 576.545,A -85,B 0,C 180,E1 -25892.244,E2 -25892.244} C_VEL
LIN {X 0,Y 112.405,Z 582.614,A -85,B 0,C 180,E1 -25897.966,E2 -25897.966} C_VEL
LIN {X 0,Y 112.319,Z 587.596,A -85,B 0,C 180,E1 -25903.645,E2 -25903.645} C_VEL
LIN {X 0,Y 112.966,Z 591.706,A -85,B 0,C 180,E1 -25909.242,E2 -25909.242} C_VEL
LIN {X 0,Y 115.23,Z 595.872,A -85,B 0,C 180,E1 -25916.503,E2 -25916.503} C_VEL
LIN {X 0,Y 119.044,Z 598.811,A -85,B 0,C 180,E1 -25923.384,E2 -25923.384} C_VEL
LIN {X 0,Y 124.397,Z 600.584,A -85,B 0,C 180,E1 -25929.757,E2 -25929.757} C_VEL
LIN {X 0,Y 131.33,Z 601.261,A -85,B 0,C 180,E1 -25935.519,E2 -25935.519} C_VEL
LIN {X 0,Y 139.529,Z 600.861,A -85,B 0,C 180,E1 -25940.645,E2 -25940.645} C_VEL
LIN {X 0,Y 148.915,Z 599.377,A -85,B 0,C 180,E1 -25945.134,E2 -25945.134} C_VEL
LIN {X 0,Y 159.337,Z 596.776,A -85,B 0,C 180,E1 -25949.024,E2 -25949.024} C_VEL
LIN {X 0,Y 170.611,Z 593.01,A -85,B 0,C 180,E1 -25952.378,E2 -25952.378} C_VEL
LIN {X 0,Y 173.576,Z 591.889,A -85,B 0,C 180,E1 -25953.134,E2 -25953.134} C_VEL
LIN {X 0,Y 174.405,Z 591.701,A -85,B 0,C 180,E1 -25954.343,E2 -25954.343} C_VEL
LIN {X 0,Y 172.615,Z 592.711,A -85,B 0,C 180,E1 -25955.483,E2 -25955.483} C_VEL
LIN {X 0,Y 161.397,Z 597.704,A -85,B 0,C 180,E1 -25958.391,E2 -25958.391} C_VEL
LIN {X 0,Y 150.901,Z 601.638,A -85,B 0,C 180,E1 -25961.827,E2 -25961.827} C_VEL
LIN {X 0,Y 141.486,Z 604.601,A -85,B 0,C 180,E1 -25965.94,E2 -25965.94} C_VEL
LIN {X 0,Y 133.075,Z 606.695,A -85,B 0,C 180,E1 -25970.674,E2 -25970.674} C_VEL
LIN {X 0,Y 125.834,Z 607.855,A -85,B 0,C 180,E1 -25976.048,E2 -25976.048} C_VEL
LIN {X 0,Y 120.104,Z 608.051,A -85,B 0,C 180,E1 -25982.088,E2 -25982.088} C_VEL
LIN {X 0,Y 116.009,Z 607.314,A -85,B 0,C 180,E1 -25988.686,E2 -25988.686} C_VEL
LIN {X 0,Y 113.795,Z 605.645,A -85,B 0,C 180,E1 -25995.698,E2 -25995.698} C_VEL
LIN {X 0,Y 113.322,Z 602.862,A -85,B 0,C 180,E1 -26002.875,E2 -26002.875} C_VEL
LIN {X 0,Y 113.696,Z 599.914,A -85,B 0,C 180,E1 -26008.229,E2 -26008.229} C_VEL
LIN {X 0,Y 113.752,Z 597.378,A -85,B 0,C 180,E1 -26011.77,E2 -26011.77} C_VEL
LIN {X 0,Y 113.731,Z 592.641,A -85,B 0,C 180,E1 -26017.099,E2 -26017.099} C_VEL
LIN {X 0,Y 114.362,Z 585.674,A -85,B 0,C 180,E1 -26023.324,E2 -26023.324} C_VEL
LIN {X 0,Y 115.895,Z 576.976,A -85,B 0,C 180,E1 -26029.483,E2 -26029.483} C_VEL
LIN {X 0,Y 118.306,Z 568.058,A -85,B 0,C 180,E1 -26034.571,E2 -26034.571} C_VEL
LIN {X 0,Y 121.584,Z 556.716,A -85,B 0,C 180,E1 -26039.672,E2 -26039.672} C_VEL
LIN {X 0,Y 123.357,Z 551.029,A -85,B 0,C 180,E1 -26041.802,E2 -26041.802} C_VEL
LIN {X 0,Y 123.1,Z 539.062,A -85,B 0,C 180,E1 -26045.94,E2 -26045.94} C_VEL
LIN {X 0,Y 122.726,Z 527.212,A -85,B 0,C 180,E1 -26049.46,E2 -26049.46} C_VEL
LIN {X 0,Y 122.133,Z 514.092,A -85,B 0,C 180,E1 -26052.805,E2 -26052.805} C_VEL
LIN {X 0,Y 121.194,Z 501.123,A -85,B 0,C 180,E1 -26055.626,E2 -26055.626} C_VEL
LIN {X 0,Y 119.313,Z 493.384,A -85,B 0,C 180,E1 -26057.347,E2 -26057.347} C_VEL
LIN {X 0,Y 115.647,Z 481.84,A -85,B 0,C 180,E1 -26059.927,E2 -26059.927} C_VEL
LIN {X 0,Y 115.597,Z 481.393,A -85,B 0,C 180,E1 -26060.049,E2 -26060.049} C_VEL
LIN {X 0,Y 115.332,Z 479.747,A -85,B 0,C 180,E1 -26063.55,E2 -26063.55} C_VEL
LIN {X 0,Y 114.938,Z 479.795,A -85,B 0,C 180,E1 -26070.715,E2 -26070.715} C_VEL
LIN {X 0,Y 114.981,Z 479.786,A -85,B 0,C 180,E1 -26078.486,E2 -26078.486} C_VEL
LIN {X 0,Y 115.147,Z 479.763,A -85,B 0,C 180,E1 -26085.87,E2 -26085.87} C_VEL
LIN {X 0,Y 115.362,Z 479.739,A -85,B 0,C 180,E1 -26089.47,E2 -26089.47} C_VEL
LIN {X 0,Y 115.575,Z 479.709,A -85,B 0,C 180,E1 -26097.068,E2 -26097.068} C_VEL
LIN {X 0,Y 115.383,Z 479.736,A -85,B 0,C 180,E1 -26099.009,E2 -26099.009} C_VEL
LIN {X 0,Y 114.079,Z 479.895,A -85,B 0,C 180,E1 -26101.887,E2 -26101.887} C_VEL
LIN {X 0,Y 108.578,Z 480.578,A -85,B 0,C 180,E1 -26110.823,E2 -26110.823} C_VEL
LIN {X 0,Y 108.199,Z 480.631,A -85,B 0,C 180,E1 -26112.962,E2 -26112.962} C_VEL
LIN {X 0,Y 107.904,Z 480.661,A -85,B 0,C 180,E1 -26119.006,E2 -26119.006} C_VEL
LIN {X 0,Y 107.857,Z 480.676,A -85,B 0,C 180,E1 -26124.185,E2 -26124.185} C_VEL
LIN {X 0,Y 107.794,Z 480.683,A -85,B 0,C 180,E1 -26132.053,E2 -26132.053} C_VEL
LIN {X 0,Y 107.708,Z 480.688,A -85,B 0,C 180,E1 -26138.465,E2 -26138.465} C_VEL
LIN {X 0,Y 107.686,Z 480.689,A -85,B 0,C 180,E1 -26145.883,E2 -26145.883} C_VEL
LIN {X 0,Y 107.71,Z 480.693,A -85,B 0,C 180,E1 -26151.537,E2 -26151.537} C_VEL
LIN {X 0,Y 107.809,Z 480.681,A -85,B 0,C 180,E1 -26158.567,E2 -26158.567} C_VEL
LIN {X 0,Y 107.913,Z 480.667,A -85,B 0,C 180,E1 -26166.999,E2 -26166.999} C_VEL
LIN {X 0,Y 108.033,Z 480.651,A -85,B 0,C 180,E1 -26174.917,E2 -26174.917} C_VEL
LIN {X 0,Y 108.255,Z 480.623,A -85,B 0,C 180,E1 -26178.769,E2 -26178.769} C_VEL
LIN {X 0,Y 108.446,Z 480.601,A -85,B 0,C 180,E1 -26186.284,E2 -26186.284} C_VEL
LIN {X 0,Y 108.945,Z 480.532,A -85,B 0,C 180,E1 -26190,E2 -26190} C_VEL
LIN {X 0,Y 108.309,Z 480.612,A -85,B 0,C 180,E1 -26197.457,E2 -26197.457} C_VEL
LIN {X 0,Y 108.176,Z 480.635,A -85,B 0,C 180,E1 -26202.956,E2 -26202.956} C_VEL
LIN {X 0,Y 107.926,Z 480.666,A -85,B 0,C 180,E1 -26211.989,E2 -26211.989} C_VEL
LIN {X 0,Y 108.17,Z 481.815,A -85,B 0,C 180,E1 -26212.439,E2 -26212.439} C_VEL
LIN {X 0,Y 112.569,Z 493.228,A -85,B 0,C 180,E1 -26215.914,E2 -26215.914} C_VEL
LIN {X 0,Y 116.145,Z 504.602,A -85,B 0,C 180,E1 -26219.448,E2 -26219.448} C_VEL
LIN {X 0,Y 119.174,Z 516.591,A -85,B 0,C 180,E1 -26223.309,E2 -26223.309} C_VEL
LIN {X 0,Y 120.479,Z 523.68,A -85,B 0,C 180,E1 -26225.685,E2 -26225.685} C_VEL
LIN {X 0,Y 119.189,Z 528.812,A -85,B 0,C 180,E1 -26227.246,E2 -26227.246} C_VEL
LIN {X 0,Y 115.543,Z 540.62,A -85,B 0,C 180,E1 -26231.371,E2 -26231.371} C_VEL
LIN {X 0,Y 112.042,Z 551.927,A -85,B 0,C 180,E1 -26236.37,E2 -26236.37} C_VEL
LIN {X 0,Y 109.01,Z 562.442,A -85,B 0,C 180,E1 -26242.23,E2 -26242.23} C_VEL
LIN {X 0,Y 107.042,Z 571.133,A -85,B 0,C 180,E1 -26248.314,E2 -26248.314} C_VEL
LIN {X 0,Y 105.66,Z 579.29,A -85,B 0,C 180,E1 -26255.434,E2 -26255.434} C_VEL
LIN {X 0,Y 105.228,Z 585.77,A -85,B 0,C 180,E1 -26262.509,E2 -26262.509} C_VEL
LIN {X 0,Y 106.136,Z 591.507,A -85,B 0,C 180,E1 -26270.455,E2 -26270.455} C_VEL
LIN {X 0,Y 107.896,Z 594.889,A -85,B 0,C 180,E1 -26276.265,E2 -26276.265} C_VEL
LIN {X 0,Y 111.71,Z 598.287,A -85,B 0,C 180,E1 -26283.606,E2 -26283.606} C_VEL
LIN {X 0,Y 117.18,Z 600.548,A -85,B 0,C 180,E1 -26290.365,E2 -26290.365} C_VEL
LIN {X 0,Y 124.843,Z 601.755,A -85,B 0,C 180,E1 -26296.864,E2 -26296.864} C_VEL
LIN {X 0,Y 132.686,Z 601.79,A -85,B 0,C 180,E1 -26301.763,E2 -26301.763} C_VEL
LIN {X 0,Y 142.342,Z 600.806,A -85,B 0,C 180,E1 -26306.382,E2 -26306.382} C_VEL
LIN {X 0,Y 153.016,Z 598.732,A -85,B 0,C 180,E1 -26310.346,E2 -26310.346} C_VEL
LIN {X 0,Y 165.273,Z 595.306,A -85,B 0,C 180,E1 -26313.933,E2 -26313.933} C_VEL
LIN {X 0,Y 164.154,Z 595.814,A -85,B 0,C 180,E1 -26314.574,E2 -26314.574} C_VEL
LIN {X 0,Y 151.572,Z 600.434,A -85,B 0,C 180,E1 -26317.98,E2 -26317.98} C_VEL
LIN {X 0,Y 141.289,Z 603.547,A -85,B 0,C 180,E1 -26321.745,E2 -26321.745} C_VEL
LIN {X 0,Y 131.916,Z 605.759,A -85,B 0,C 180,E1 -26326.166,E2 -26326.166} C_VEL
LIN {X 0,Y 123.658,Z 607.051,A -85,B 0,C 180,E1 -26331.306,E2 -26331.306} C_VEL
LIN {X 0,Y 115.48,Z 607.423,A -85,B 0,C 180,E1 -26338.432,E2 -26338.432} C_VEL
LIN {X 0,Y 111.456,Z 606.981,A -85,B 0,C 180,E1 -26343.808,E2 -26343.808} C_VEL
LIN {X 0,Y 107.951,Z 605.496,A -85,B 0,C 180,E1 -26351.003,E2 -26351.003} C_VEL
LIN {X 0,Y 106.467,Z 603.049,A -85,B 0,C 180,E1 -26358.578,E2 -26358.578} C_VEL
LIN {X 0,Y 106.396,Z 601.407,A -85,B 0,C 180,E1 -26362.409,E2 -26362.409} C_VEL
LIN {X 0,Y 106.792,Z 598.315,A -85,B 0,C 180,E1 -26368.114,E2 -26368.114} C_VEL
LIN {X 0,Y 106.797,Z 595.646,A -85,B 0,C 180,E1 -26371.886,E2 -26371.886} C_VEL
LIN {X 0,Y 106.776,Z 590.66,A -85,B 0,C 180,E1 -26377.564,E2 -26377.564} C_VEL
LIN {X 0,Y 107.539,Z 583.367,A -85,B 0,C 180,E1 -26384.186,E2 -26384.186} C_VEL
LIN {X 0,Y 109.309,Z 574.316,A -85,B 0,C 180,E1 -26390.709,E2 -26390.709} C_VEL
LIN {X 0,Y 111.956,Z 564.995,A -85,B 0,C 180,E1 -26396.067,E2 -26396.067} C_VEL
LIN {X 0,Y 115.154,Z 554.439,A -85,B 0,C 180,E1 -26400.903,E2 -26400.903} C_VEL
LIN {X 0,Y 116.288,Z 550.736,A -85,B 0,C 180,E1 -26402.349,E2 -26402.349} C_VEL
LIN {X 0,Y 116.107,Z 538.839,A -85,B 0,C 180,E1 -26406.707,E2 -26406.707} C_VEL
LIN {X 0,Y 115.806,Z 527.469,A -85,B 0,C 180,E1 -26410.289,E2 -26410.289} C_VEL
LIN {X 0,Y 115.293,Z 513.351,A -85,B 0,C 180,E1 -26414.099,E2 -26414.099} C_VEL
LIN {X 0,Y 114.417,Z 501.839,A -85,B 0,C 180,E1 -26416.82,E2 -26416.82} C_VEL
LIN {X 0,Y 111.54,Z 491.146,A -85,B 0,C 180,E1 -26419.475,E2 -26419.475} C_VEL
LIN {X 0,Y 108.382,Z 481.361,A -85,B 0,C 180,E1 -26421.89,E2 -26421.89} C_VEL
LIN {X 0,Y 108.313,Z 480.933,A -85,B 0,C 180,E1 -26422.036,E2 -26422.036} C_VEL
LIN {X 0,Y 108.292,Z 480.624,A -85,B 0,C 180,E1 -26423.153,E2 -26423.153} C_VEL
LIN {X 0,Y 107.98,Z 480.661,A -85,B 0,C 180,E1 -26428.622,E2 -26428.622} C_VEL
LIN {X 0,Y 107.91,Z 480.663,A -85,B 0,C 180,E1 -26436.998,E2 -26436.998} C_VEL
LIN {X 0,Y 108.039,Z 480.645,A -85,B 0,C 180,E1 -26444.919,E2 -26444.919} C_VEL
LIN {X 0,Y 108.287,Z 480.622,A -85,B 0,C 180,E1 -26448.773,E2 -26448.773} C_VEL
LIN {X 0,Y 108.456,Z 480.599,A -85,B 0,C 180,E1 -26456.285,E2 -26456.285} C_VEL
LIN {X 0,Y 108.944,Z 480.537,A -85,B 0,C 180,E1 -26460.001,E2 -26460.001} C_VEL
LIN {X 0,Y 108.328,Z 480.615,A -85,B 0,C 180,E1 -26467.456,E2 -26467.456} C_VEL
LIN {X 0,Y 108.199,Z 480.631,A -85,B 0,C 180,E1 -26472.962,E2 -26472.962} C_VEL
LIN {X 0,Y 107.456,Z 480.739,A -85,B 0,C 180,E1 -26476.062,E2 -26476.062} C_VEL
LIN {X 0,Y 105.798,Z 480.952,A -85,B 0,C 180,E1 -26479.125,E2 -26479.125} C_VEL
LIN {X 0,Y 101.011,Z 481.526,A -85,B 0,C 180,E1 -26487.674,E2 -26487.674} C_VEL
LIN {X 0,Y 100.636,Z 481.565,A -85,B 0,C 180,E1 -26489.963,E2 -26489.963} C_VEL
LIN {X 0,Y 100.676,Z 481.569,A -85,B 0,C 180,E1 -26493.951,E2 -26493.951} C_VEL
LIN {X 0,Y 100.655,Z 481.57,A -85,B 0,C 180,E1 -26499.822,E2 -26499.822} C_VEL
LIN {X 0,Y 100.656,Z 481.564,A -85,B 0,C 180,E1 -26505.717,E2 -26505.717} C_VEL
LIN {X 0,Y 100.647,Z 481.572,A -85,B 0,C 180,E1 -26511.065,E2 -26511.065} C_VEL
LIN {X 0,Y 100.702,Z 481.564,A -85,B 0,C 180,E1 -26516.877,E2 -26516.877} C_VEL
LIN {X 0,Y 100.788,Z 481.551,A -85,B 0,C 180,E1 -26525.268,E2 -26525.268} C_VEL
LIN {X 0,Y 100.818,Z 481.55,A -85,B 0,C 180,E1 -26529.602,E2 -26529.602} C_VEL
LIN {X 0,Y 101.103,Z 481.516,A -85,B 0,C 180,E1 -26536.707,E2 -26536.707} C_VEL
LIN {X 0,Y 101.243,Z 481.492,A -85,B 0,C 180,E1 -26542.02,E2 -26542.02} C_VEL
LIN {X 0,Y 101.868,Z 481.413,A -85,B 0,C 180,E1 -26550,E2 -26550} C_VEL
LIN {X 0,Y 101.247,Z 481.491,A -85,B 0,C 180,E1 -26557.98,E2 -26557.98} C_VEL
LIN {X 0,Y 101.105,Z 481.517,A -85,B 0,C 180,E1 -26563.298,E2 -26563.298} C_VEL
LIN {X 0,Y 100.858,Z 481.548,A -85,B 0,C 180,E1 -26570.257,E2 -26570.257} C_VEL
LIN {X 0,Y 105.879,Z 494.988,A -85,B 0,C 180,E1 -26574.744,E2 -26574.744} C_VEL
LIN {X 0,Y 109.316,Z 505.821,A -85,B 0,C 180,E1 -26578.36,E2 -26578.36} C_VEL
LIN {X 0,Y 112.355,Z 518.144,A -85,B 0,C 180,E1 -26582.65,E2 -26582.65} C_VEL
LIN {X 0,Y 113.445,Z 523.921,A -85,B 0,C 180,E1 -26584.748,E2 -26584.748} C_VEL
LIN {X 0,Y 113.211,Z 525.962,A -85,B 0,C 180,E1 -26585.432,E2 -26585.432} C_VEL
LIN {X 0,Y 108.912,Z 539.435,A -85,B 0,C 180,E1 -26590.187,E2 -26590.187} C_VEL
LIN {X 0,Y 105.525,Z 549.987,A -85,B 0,C 180,E1 -26594.957,E2 -26594.957} C_VEL
LIN {X 0,Y 102.454,Z 560.064,A -85,B 0,C 180,E1 -26600.679,E2 -26600.679} C_VEL
LIN {X 0,Y 100.226,Z 569.41,A -85,B 0,C 180,E1 -26607.293,E2 -26607.293} C_VEL
LIN {X 0,Y 98.683,Z 577.766,A -85,B 0,C 180,E1 -26614.702,E2 -26614.702} C_VEL
LIN {X 0,Y 98.188,Z 583.67,A -85,B 0,C 180,E1 -26621.209,E2 -26621.209} C_VEL
LIN {X 0,Y 98.896,Z 589.985,A -85,B 0,C 180,E1 -26629.766,E2 -26629.766} C_VEL
LIN {X 0,Y 101.365,Z 594.815,A -85,B 0,C 180,E1 -26638.013,E2 -26638.013} C_VEL
LIN {X 0,Y 106.982,Z 599.059,A -85,B 0,C 180,E1 -26647.549,E2 -26647.549} C_VEL
LIN {X 0,Y 113.379,Z 601.229,A -85,B 0,C 180,E1 -26654.355,E2 -26654.355} C_VEL
LIN {X 0,Y 121.381,Z 602.352,A -85,B 0,C 180,E1 -26660.328,E2 -26660.328} C_VEL
LIN {X 0,Y 130.735,Z 602.397,A -85,B 0,C 180,E1 -26665.471,E2 -26665.471} C_VEL
LIN {X 0,Y 141.16,Z 601.378,A -85,B 0,C 180,E1 -26669.859,E2 -26669.859} C_VEL
LIN {X 0,Y 152.494,Z 599.308,A -85,B 0,C 180,E1 -26673.576,E2 -26673.576} C_VEL
LIN {X 0,Y 153.038,Z 599.274,A -85,B 0,C 180,E1 -26674.249,E2 -26674.249} C_VEL
LIN {X 0,Y 141.855,Z 602.52,A -85,B 0,C 180,E1 -26677.563,E2 -26677.563} C_VEL
LIN {X 0,Y 131.637,Z 604.8,A -85,B 0,C 180,E1 -26681.631,E2 -26681.631} C_VEL
LIN {X 0,Y 122.386,Z 606.253,A -85,B 0,C 180,E1 -26686.442,E2 -26686.442} C_VEL
LIN {X 0,Y 114.317,Z 606.848,A -85,B 0,C 180,E1 -26692.065,E2 -26692.065} C_VEL
LIN {X 0,Y 107.719,Z 606.502,A -85,B 0,C 180,E1 -26698.538,E2 -26698.538} C_VEL
LIN {X 0,Y 102.949,Z 605.264,A -85,B 0,C 180,E1 -26705.821,E2 -26705.821} C_VEL
LIN {X 0,Y 100.231,Z 603.122,A -85,B 0,C 180,E1 -26713.712,E2 -26713.712} C_VEL
LIN {X 0,Y 99.51,Z 599.204,A -85,B 0,C 180,E1 -26723.288,E2 -26723.288} C_VEL
LIN {X 0,Y 99.894,Z 596.61,A -85,B 0,C 180,E1 -26727.984,E2 -26727.984} C_VEL
LIN {X 0,Y 99.875,Z 593.767,A -85,B 0,C 180,E1 -26732.016,E2 -26732.016} C_VEL
LIN {X 0,Y 99.937,Z 587.456,A -85,B 0,C 180,E1 -26739.191,E2 -26739.191} C_VEL
LIN {X 0,Y 100.734,Z 580.954,A -85,B 0,C 180,E1 -26745.166,E2 -26745.166} C_VEL
LIN {X 0,Y 102.391,Z 573.005,A -85,B 0,C 180,E1 -26751.121,E2 -26751.121} C_VEL
LIN {X 0,Y 105.15,Z 563.506,A -85,B 0,C 180,E1 -26756.817,E2 -26756.817} C_VEL
LIN {X 0,Y 108.79,Z 551.981,A -85,B 0,C 180,E1 -26762.245,E2 -26762.245} C_VEL
LIN {X 0,Y 109.229,Z 549.627,A -85,B 0,C 180,E1 -26763.235,E2 -26763.235} C_VEL
LIN {X 0,Y 109.131,Z 538.052,A -85,B 0,C 180,E1 -26767.719,E2 -26767.719} C_VEL
LIN {X 0,Y 108.855,Z 524.954,A -85,B 0,C 180,E1 -26772.054,E2 -26772.054} C_VEL
LIN {X 0,Y 108.366,Z 510.247,A -85,B 0,C 180,E1 -26776.175,E2 -26776.175} C_VEL
LIN {X 0,Y 107.659,Z 502.524,A -85,B 0,C 180,E1 -26778.158,E2 -26778.158} C_VEL
LIN {X 0,Y 104.265,Z 490.638,A -85,B 0,C 180,E1 -26781.402,E2 -26781.402} C_VEL
LIN {X 0,Y 101.24,Z 481.5,A -85,B 0,C 180,E1 -26783.993,E2 -26783.993} C_VEL
LIN {X 0,Y 100.79,Z 481.557,A -85,B 0,C 180,E1 -26790.785,E2 -26790.785} C_VEL
LIN {X 0,Y 100.785,Z 481.545,A -85,B 0,C 180,E1 -26795.267,E2 -26795.267} C_VEL
LIN {X 0,Y 100.818,Z 481.551,A -85,B 0,C 180,E1 -26799.602,E2 -26799.602} C_VEL
LIN {X 0,Y 101.186,Z 481.505,A -85,B 0,C 180,E1 -26807.974,E2 -26807.974} C_VEL
LIN {X 0,Y 101.266,Z 481.49,A -85,B 0,C 180,E1 -26812.022,E2 -26812.022} C_VEL
LIN {X 0,Y 101.868,Z 481.418,A -85,B 0,C 180,E1 -26820.001,E2 -26820.001} C_VEL
LIN {X 0,Y 101.267,Z 481.495,A -85,B 0,C 180,E1 -26827.979,E2 -26827.979} C_VEL
LIN {X 0,Y 101.124,Z 481.512,A -85,B 0,C 180,E1 -26833.352,E2 -26833.352} C_VEL
LIN {X 0,Y 100.815,Z 481.545,A -85,B 0,C 180,E1 -26840.4,E2 -26840.4} C_VEL
LIN {X 0,Y 100.774,Z 481.556,A -85,B 0,C 180,E1 -26844.96,E2 -26844.96} C_VEL
LIN {X 0,Y 100.636,Z 481.565,A -85,B 0,C 180,E1 -26849.963,E2 -26849.963} C_VEL
LIN {X 0,Y 99.9,Z 481.666,A -85,B 0,C 180,E1 -26853.305,E2 -26853.305} C_VEL
LIN {X 0,Y 98.299,Z 481.864,A -85,B 0,C 180,E1 -26856.616,E2 -26856.616} C_VEL
LIN {X 0,Y 93.822,Z 482.418,A -85,B 0,C 180,E1 -26865.886,E2 -26865.886} C_VEL
LIN {X 0,Y 93.541,Z 482.455,A -85,B 0,C 180,E1 -26868.356,E2 -26868.356} C_VEL
LIN {X 0,Y 93.6,Z 482.444,A -85,B 0,C 180,E1 -26875.686,E2 -26875.686} C_VEL
LIN {X 0,Y 93.671,Z 482.435,A -85,B 0,C 180,E1 -26884.205,E2 -26884.205} C_VEL
LIN {X 0,Y 93.695,Z 482.439,A -85,B 0,C 180,E1 -26887.973,E2 -26887.973} C_VEL
LIN {X 0,Y 94.023,Z 482.398,A -85,B 0,C 180,E1 -26896.346,E2 -26896.346} C_VEL
LIN {X 0,Y 94.177,Z 482.371,A -85,B 0,C 180,E1 -26901.417,E2 -26901.417} C_VEL
LIN {X 0,Y 94.794,Z 482.294,A -85,B 0,C 180,E1 -26910,E2 -26910} C_VEL
LIN {X 0,Y 94.18,Z 482.368,A -85,B 0,C 180,E1 -26918.583,E2 -26918.583} C_VEL
LIN {X 0,Y 94.02,Z 482.401,A -85,B 0,C 180,E1 -26923.647,E2 -26923.647} C_VEL
LIN {X 0,Y 93.884,Z 482.617,A -85,B 0,C 180,E1 -26928.268,E2 -26928.268} C_VEL
LIN {X 0,Y 98.374,Z 494.302,A -85,B 0,C 180,E1 -26932.581,E2 -26932.581} C_VEL
LIN {X 0,Y 101.945,Z 505.322,A -85,B 0,C 180,E1 -26936.622,E2 -26936.622} C_VEL
LIN {X 0,Y 105.068,Z 517.738,A -85,B 0,C 180,E1 -26941.224,E2 -26941.224} C_VEL
LIN {X 0,Y 106.563,Z 525.164,A -85,B 0,C 180,E1 -26944.096,E2 -26944.096} C_VEL
LIN {X 0,Y 102.434,Z 537.795,A -85,B 0,C 180,E1 -26948.74,E2 -26948.74} C_VEL
LIN {X 0,Y 98.443,Z 549.834,A -85,B 0,C 180,E1 -26954.444,E2 -26954.444} C_VEL
LIN {X 0,Y 95.085,Z 560.755,A -85,B 0,C 180,E1 -26961.077,E2 -26961.077} C_VEL
LIN {X 0,Y 92.893,Z 569.82,A -85,B 0,C 180,E1 -26968.02,E2 -26968.02} C_VEL
LIN {X 0,Y 91.508,Z 578.258,A -85,B 0,C 180,E1 -26976.22,E2 -26976.22} C_VEL
LIN {X 0,Y 91.226,Z 584.975,A -85,B 0,C 180,E1 -26984.356,E2 -26984.356} C_VEL
LIN {X 0,Y 92.262,Z 590.13,A -85,B 0,C 180,E1 -26991.994,E2 -26991.994} C_VEL
LIN {X 0,Y 94.949,Z 594.611,A -85,B 0,C 180,E1 -26999.999,E2 -26999.999} C_VEL
LIN {X 0,Y 99.73,Z 598.355,A -85,B 0,C 180,E1 -27008.102,E2 -27008.102} C_VEL
LIN {X 0,Y 106.289,Z 600.977,A -85,B 0,C 180,E1 -27015.336,E2 -27015.336} C_VEL
LIN {X 0,Y 114.514,Z 602.568,A -85,B 0,C 180,E1 -27021.606,E2 -27021.606} C_VEL
LIN {X 0,Y 124.121,Z 603.128,A -85,B 0,C 180,E1 -27026.934,E2 -27026.934} C_VEL
LIN {X 0,Y 134.818,Z 602.633,A -85,B 0,C 180,E1 -27031.419,E2 -27031.419} C_VEL
LIN {X 0,Y 141.369,Z 601.884,A -85,B 0,C 180,E1 -27033.627,E2 -27033.627} C_VEL
LIN {X 0,Y 140.628,Z 602.117,A -85,B 0,C 180,E1 -27034.31,E2 -27034.31} C_VEL
LIN {X 0,Y 127.028,Z 604.763,A -85,B 0,C 180,E1 -27039.236,E2 -27039.236} C_VEL
LIN {X 0,Y 117.333,Z 605.917,A -85,B 0,C 180,E1 -27044.048,E2 -27044.048} C_VEL
LIN {X 0,Y 108.812,Z 606.175,A -85,B 0,C 180,E1 -27049.769,E2 -27049.769} C_VEL
LIN {X 0,Y 101.729,Z 605.584,A -85,B 0,C 180,E1 -27056.45,E2 -27056.45} C_VEL
LIN {X 0,Y 96.575,Z 604.13,A -85,B 0,C 180,E1 -27064.111,E2 -27064.111} C_VEL
LIN {X 0,Y 93.531,Z 601.702,A -85,B 0,C 180,E1 -27072.509,E2 -27072.509} C_VEL
LIN {X 0,Y 92.661,Z 597.713,A -85,B 0,C 180,E1 -27082.392,E2 -27082.392} C_VEL
LIN {X 0,Y 93.024,Z 594.818,A -85,B 0,C 180,E1 -27087.835,E2 -27087.835} C_VEL
LIN {X 0,Y 92.942,Z 591.856,A -85,B 0,C 180,E1 -27092.167,E2 -27092.167} C_VEL
LIN {X 0,Y 93.001,Z 585.629,A -85,B 0,C 180,E1 -27099.413,E2 -27099.413} C_VEL
LIN {X 0,Y 93.935,Z 578.302,A -85,B 0,C 180,E1 -27106.294,E2 -27106.294} C_VEL
LIN {X 0,Y 96.321,Z 568.516,A -85,B 0,C 180,E1 -27113.659,E2 -27113.659} C_VEL
LIN {X 0,Y 99.486,Z 558.327,A -85,B 0,C 180,E1 -27119.636,E2 -27119.636} C_VEL
LIN {X 0,Y 102.126,Z 550.348,A -85,B 0,C 180,E1 -27123.403,E2 -27123.403} C_VEL
LIN {X 0,Y 102.159,Z 538.825,A -85,B 0,C 180,E1 -27128.253,E2 -27128.253} C_VEL
LIN {X 0,Y 101.979,Z 525.152,A -85,B 0,C 180,E1 -27133.144,E2 -27133.144} C_VEL
LIN {X 0,Y 101.63,Z 510.204,A -85,B 0,C 180,E1 -27137.606,E2 -27137.606} C_VEL
LIN {X 0,Y 101.021,Z 504.161,A -85,B 0,C 180,E1 -27139.292,E2 -27139.292} C_VEL
LIN {X 0,Y 97.308,Z 490.961,A -85,B 0,C 180,E1 -27143.299,E2 -27143.299} C_VEL
LIN {X 0,Y 95.324,Z 485.566,A -85,B 0,C 180,E1 -27145.023,E2 -27145.023} C_VEL
LIN {X 0,Y 94.176,Z 483.123,A -85,B 0,C 180,E1 -27145.882,E2 -27145.882} C_VEL
LIN {X 0,Y 94.016,Z 482.393,A -85,B 0,C 180,E1 -27146.171,E2 -27146.171} C_VEL
LIN {X 0,Y 93.703,Z 482.426,A -85,B 0,C 180,E1 -27154.161,E2 -27154.161} C_VEL
LIN {X 0,Y 93.694,Z 482.437,A -85,B 0,C 180,E1 -27157.973,E2 -27157.973} C_VEL
LIN {X 0,Y 94.09,Z 482.388,A -85,B 0,C 180,E1 -27167.052,E2 -27167.052} C_VEL
LIN {X 0,Y 94.198,Z 482.372,A -85,B 0,C 180,E1 -27171.419,E2 -27171.419} C_VEL
LIN {X 0,Y 94.794,Z 482.298,A -85,B 0,C 180,E1 -27180.001,E2 -27180.001} C_VEL
LIN {X 0,Y 94.199,Z 482.372,A -85,B 0,C 180,E1 -27188.582,E2 -27188.582} C_VEL
LIN {X 0,Y 94.042,Z 482.394,A -85,B 0,C 180,E1 -27193.71,E2 -27193.71} C_VEL
LIN {X 0,Y 93.693,Z 482.437,A -85,B 0,C 180,E1 -27202.029,E2 -27202.029} C_VEL
LIN {X 0,Y 93.623,Z 482.443,A -85,B 0,C 180,E1 -27206.771,E2 -27206.771} C_VEL
LIN {X 0,Y 93.598,Z 482.449,A -85,B 0,C 180,E1 -27214.316,E2 -27214.316} C_VEL
LIN {X 0,Y 93.542,Z 482.457,A -85,B 0,C 180,E1 -27222.548,E2 -27222.548} C_VEL
LIN {X 0,Y 93.541,Z 482.455,A -85,B 0,C 180,E1 -27228.356,E2 -27228.356} C_VEL
LIN {X 0,Y 93.249,Z 482.5,A -85,B 0,C 180,E1 -27230.758,E2 -27230.758} C_VEL
LIN {X 0,Y 92.46,Z 482.603,A -85,B 0,C 180,E1 -27233.138,E2 -27233.138} C_VEL
LIN {X 0,Y 90.083,Z 482.899,A -85,B 0,C 180,E1 -27237.899,E2 -27237.899} C_VEL
LIN {X 0,Y 86.836,Z 483.289,A -85,B 0,C 180,E1 -27245.54,E2 -27245.54} C_VEL
LIN {X 0,Y 86.533,Z 483.317,A -85,B 0,C 180,E1 -27248.22,E2 -27248.22} C_VEL
LIN {X 0,Y 86.933,Z 483.282,A -85,B 0,C 180,E1 -27255.964,E2 -27255.964} C_VEL
LIN {X 0,Y 87.086,Z 483.254,A -85,B 0,C 180,E1 -27260.712,E2 -27260.712} C_VEL
LIN {X 0,Y 87.72,Z 483.175,A -85,B 0,C 180,E1 -27270,E2 -27270} C_VEL
LIN {X 0,Y 87.088,Z 483.249,A -85,B 0,C 180,E1 -27279.288,E2 -27279.288} C_VEL
LIN {X 0,Y 86.817,Z 483.297,A -85,B 0,C 180,E1 -27285.855,E2 -27285.855} C_VEL
LIN {X 0,Y 91.485,Z 495.428,A -85,B 0,C 180,E1 -27290.811,E2 -27290.811} C_VEL
LIN {X 0,Y 95.041,Z 506.223,A -85,B 0,C 180,E1 -27295.162,E2 -27295.162} C_VEL
LIN {X 0,Y 97.748,Z 517.263,A -85,B 0,C 180,E1 -27299.623,E2 -27299.623} C_VEL
LIN {X 0,Y 99.544,Z 525.453,A -85,B 0,C 180,E1 -27303.068,E2 -27303.068} C_VEL
LIN {X 0,Y 95.552,Z 537.512,A -85,B 0,C 180,E1 -27307.749,E2 -27307.749} C_VEL
LIN {X 0,Y 91.366,Z 549.613,A -85,B 0,C 180,E1 -27313.811,E2 -27313.811} C_VEL
LIN {X 0,Y 88.144,Z 559.756,A -85,B 0,C 180,E1 -27320.366,E2 -27320.366} C_VEL
LIN {X 0,Y 85.871,Z 568.933,A -85,B 0,C 180,E1 -27327.859,E2 -27327.859} C_VEL
LIN {X 0,Y 84.493,Z 577.129,A -85,B 0,C 180,E1 -27336.198,E2 -27336.198} C_VEL
LIN {X 0,Y 84.283,Z 584.436,A -85,B 0,C 180,E1 -27345.512,E2 -27345.512} C_VEL
LIN {X 0,Y 86,Z 590.648,A -85,B 0,C 180,E1 -27355.312,E2 -27355.312} C_VEL
LIN {X 0,Y 89.774,Z 595.469,A -85,B 0,C 180,E1 -27364.489,E2 -27364.489} C_VEL
LIN {X 0,Y 95.64,Z 599.101,A -85,B 0,C 180,E1 -27372.735,E2 -27372.735} C_VEL
LIN {X 0,Y 103.29,Z 601.661,A -85,B 0,C 180,E1 -27379.889,E2 -27379.889} C_VEL
LIN {X 0,Y 112.467,Z 603.211,A -85,B 0,C 180,E1 -27385.939,E2 -27385.939} C_VEL
LIN {X 0,Y 122.938,Z 603.757,A -85,B 0,C 180,E1 -27390.964,E2 -27390.964} C_VEL
LIN {X 0,Y 129.602,Z 603.575,A -85,B 0,C 180,E1 -27393.496,E2 -27393.496} C_VEL
LIN {X 0,Y 128.097,Z 603.911,A -85,B 0,C 180,E1 -27394.618,E2 -27394.618} C_VEL
LIN {X 0,Y 117.442,Z 605.126,A -85,B 0,C 180,E1 -27398.928,E2 -27398.928} C_VEL
LIN {X 0,Y 107.836,Z 605.537,A -85,B 0,C 180,E1 -27404.202,E2 -27404.202} C_VEL
LIN {X 0,Y 97.381,Z 604.817,A -85,B 0,C 180,E1 -27412.548,E2 -27412.548} C_VEL
LIN {X 0,Y 90.321,Z 602.844,A -85,B 0,C 180,E1 -27422.169,E2 -27422.169} C_VEL
LIN {X 0,Y 86.908,Z 600.204,A -85,B 0,C 180,E1 -27431.128,E2 -27431.128} C_VEL
LIN {X 0,Y 85.839,Z 596.561,A -85,B 0,C 180,E1 -27440.576,E2 -27440.576} C_VEL
LIN {X 0,Y 86.185,Z 592.877,A -85,B 0,C 180,E1 -27447.663,E2 -27447.663} C_VEL
LIN {X 0,Y 86.047,Z 589.713,A -85,B 0,C 180,E1 -27452.34,E2 -27452.34} C_VEL
LIN {X 0,Y 86.146,Z 583.095,A -85,B 0,C 180,E1 -27460.328,E2 -27460.328} C_VEL
LIN {X 0,Y 87.242,Z 575.583,A -85,B 0,C 180,E1 -27467.583,E2 -27467.583} C_VEL
LIN {X 0,Y 89.979,Z 565.28,A -85,B 0,C 180,E1 -27475.441,E2 -27475.441} C_VEL
LIN {X 0,Y 92.806,Z 556.483,A -85,B 0,C 180,E1 -27480.741,E2 -27480.741} C_VEL
LIN {X 0,Y 94.892,Z 550.544,A -85,B 0,C 180,E1 -27483.743,E2 -27483.743} C_VEL
LIN {X 0,Y 95.114,Z 545.257,A -85,B 0,C 180,E1 -27486.236,E2 -27486.236} C_VEL
LIN {X 0,Y 95.128,Z 534.127,A -85,B 0,C 180,E1 -27490.97,E2 -27490.97} C_VEL
LIN {X 0,Y 95.077,Z 521.001,A -85,B 0,C 180,E1 -27495.769,E2 -27495.769} C_VEL
LIN {X 0,Y 94.794,Z 507.94,A -85,B 0,C 180,E1 -27499.866,E2 -27499.866} C_VEL
LIN {X 0,Y 92.43,Z 498.196,A -85,B 0,C 180,E1 -27503.149,E2 -27503.149} C_VEL
LIN {X 0,Y 89.777,Z 489.742,A -85,B 0,C 180,E1 -27506.031,E2 -27506.031} C_VEL
LIN {X 0,Y 86.929,Z 484.107,A -85,B 0,C 180,E1 -27508.298,E2 -27508.298} C_VEL
LIN {X 0,Y 86.753,Z 483.305,A -85,B 0,C 180,E1 -27508.567,E2 -27508.567} C_VEL
LIN {X 0,Y 86.603,Z 483.313,A -85,B 0,C 180,E1 -27516.062,E2 -27516.062} C_VEL
LIN {X 0,Y 86.663,Z 483.314,A -85,B 0,C 180,E1 -27521.073,E2 -27521.073} C_VEL
LIN {X 0,Y 86.968,Z 483.273,A -85,B 0,C 180,E1 -27525.971,E2 -27525.971} C_VEL
LIN {X 0,Y 87.107,Z 483.257,A -85,B 0,C 180,E1 -27530.715,E2 -27530.715} C_VEL
LIN {X 0,Y 87.722,Z 483.179,A -85,B 0,C 180,E1 -27540.001,E2 -27540.001} C_VEL
LIN {X 0,Y 87.107,Z 483.254,A -85,B 0,C 180,E1 -27549.287,E2 -27549.287} C_VEL
LIN {X 0,Y 86.95,Z 483.278,A -85,B 0,C 180,E1 -27554.088,E2 -27554.088} C_VEL
LIN {X 0,Y 86.587,Z 483.325,A -85,B 0,C 180,E1 -27563.945,E2 -27563.945} C_VEL
LIN {X 0,Y 86.478,Z 483.331,A -85,B 0,C 180,E1 -27569.185,E2 -27569.185} C_VEL
LIN {X 0,Y 86.517,Z 483.327,A -85,B 0,C 180,E1 -27575.678,E2 -27575.678} C_VEL
LIN {X 0,Y 86.483,Z 483.336,A -85,B 0,C 180,E1 -27582.999,E2 -27582.999} C_VEL
LIN {X 0,Y 86.468,Z 483.339,A -85,B 0,C 180,E1 -27589.442,E2 -27589.442} C_VEL
LIN {X 0,Y 86.544,Z 483.321,A -85,B 0,C 180,E1 -27595.358,E2 -27595.358} C_VEL
LIN {X 0,Y 86.587,Z 483.316,A -85,B 0,C 180,E1 -27603.234,E2 -27603.234} C_VEL
LIN {X 0,Y 86.533,Z 483.317,A -85,B 0,C 180,E1 -27608.22,E2 -27608.22} C_VEL
LIN {X 0,Y 86.223,Z 483.364,A -85,B 0,C 180,E1 -27610.817,E2 -27610.817} C_VEL
LIN {X 0,Y 85.431,Z 483.461,A -85,B 0,C 180,E1 -27613.393,E2 -27613.393} C_VEL
LIN {X 0,Y 83.143,Z 483.751,A -85,B 0,C 180,E1 -27618.576,E2 -27618.576} C_VEL
LIN {X 0,Y 80.517,Z 484.079,A -85,B 0,C 180,E1 -27626.906,E2 -27626.906} C_VEL
LIN {X 0,Y 80.611,Z 484.059,A -85,B 0,C 180,E1 -27629.779,E2 -27629.779} C_VEL
LIN {X 0,Y 79.971,Z 484.136,A -85,B 0,C 180,E1 -27640.123,E2 -27640.123} C_VEL
LIN {X 0,Y 79.892,Z 484.159,A -85,B 0,C 180,E1 -27643.05,E2 -27643.05} C_VEL
LIN {X 0,Y 84.495,Z 496.148,A -85,B 0,C 180,E1 -27648.672,E2 -27648.672} C_VEL
LIN {X 0,Y 88.048,Z 507.034,A -85,B 0,C 180,E1 -27653.522,E2 -27653.522} C_VEL
LIN {X 0,Y 90.5,Z 516.747,A -85,B 0,C 180,E1 -27657.771,E2 -27657.771} C_VEL
LIN {X 0,Y 92.507,Z 526.321,A -85,B 0,C 180,E1 -27662.127,E2 -27662.127} C_VEL
LIN {X 0,Y 88.226,Z 538.404,A -85,B 0,C 180,E1 -27667.192,E2 -27667.192} C_VEL
LIN {X 0,Y 84.305,Z 549.35,A -85,B 0,C 180,E1 -27673.159,E2 -27673.159} C_VEL
LIN {X 0,Y 80.74,Z 560.508,A -85,B 0,C 180,E1 -27681.031,E2 -27681.031} C_VEL
LIN {X 0,Y 78.545,Z 569.426,A -85,B 0,C 180,E1 -27689.035,E2 -27689.035} C_VEL
LIN {X 0,Y 77.441,Z 576.42,A -85,B 0,C 180,E1 -27696.783,E2 -27696.783} C_VEL
LIN {X 0,Y 77.393,Z 583.806,A -85,B 0,C 180,E1 -27706.877,E2 -27706.877} C_VEL
LIN {X 0,Y 79.498,Z 590.211,A -85,B 0,C 180,E1 -27717.466,E2 -27717.466} C_VEL
LIN {X 0,Y 83.803,Z 595.184,A -85,B 0,C 180,E1 -27727.226,E2 -27727.226} C_VEL
LIN {X 0,Y 88.513,Z 598.188,A -85,B 0,C 180,E1 -27733.78,E2 -27733.78} C_VEL
LIN {X 0,Y 96.405,Z 601.191,A -85,B 0,C 180,E1 -27741.376,E2 -27741.376} C_VEL
LIN {X 0,Y 105.878,Z 603.208,A -85,B 0,C 180,E1 -27747.687,E2 -27747.687} C_VEL
LIN {X 0,Y 117.586,Z 604.268,A -85,B 0,C 180,E1 -27753.201,E2 -27753.201} C_VEL
LIN {X 0,Y 118.56,Z 604.347,A -85,B 0,C 180,E1 -27753.914,E2 -27753.914} C_VEL
LIN {X 0,Y 107.938,Z 604.888,A -85,B 0,C 180,E1 -27758.618,E2 -27758.618} C_VEL
LIN {X 0,Y 98.432,Z 604.576,A -85,B 0,C 180,E1 -27764.44,E2 -27764.44} C_VEL
LIN {X 0,Y 90.304,Z 603.44,A -85,B 0,C 180,E1 -27771.494,E2 -27771.494} C_VEL
LIN {X 0,Y 84.178,Z 601.49,A -85,B 0,C 180,E1 -27779.939,E2 -27779.939} C_VEL
LIN {X 0,Y 80.346,Z 598.592,A -85,B 0,C 180,E1 -27789.52,E2 -27789.52} C_VEL
LIN {X 0,Y 79.089,Z 594.666,A -85,B 0,C 180,E1 -27799.763,E2 -27799.763} C_VEL
LIN {X 0,Y 79.34,Z 590.886,A -85,B 0,C 180,E1 -27807.462,E2 -27807.462} C_VEL
LIN {X 0,Y 79.14,Z 587.53,A -85,B 0,C 180,E1 -27812.545,E2 -27812.545} C_VEL
LIN {X 0,Y 79.239,Z 581.401,A -85,B 0,C 180,E1 -27820.217,E2 -27820.217} C_VEL
LIN {X 0,Y 80.322,Z 574.01,A -85,B 0,C 180,E1 -27827.833,E2 -27827.833} C_VEL
LIN {X 0,Y 82.672,Z 565.243,A -85,B 0,C 180,E1 -27835.153,E2 -27835.153} C_VEL
LIN {X 0,Y 85.534,Z 556.568,A -85,B 0,C 180,E1 -27840.899,E2 -27840.899} C_VEL
LIN {X 0,Y 88.083,Z 548.861,A -85,B 0,C 180,E1 -27845.089,E2 -27845.089} C_VEL
LIN {X 0,Y 88.2,Z 536.379,A -85,B 0,C 180,E1 -27851.099,E2 -27851.099} C_VEL
LIN {X 0,Y 88.302,Z 522.711,A -85,B 0,C 180,E1 -27856.643,E2 -27856.643} C_VEL
LIN {X 0,Y 88.233,Z 509.651,A -85,B 0,C 180,E1 -27861.152,E2 -27861.152} C_VEL
LIN {X 0,Y 86.129,Z 500.762,A -85,B 0,C 180,E1 -27864.453,E2 -27864.453} C_VEL
LIN {X 0,Y 83.976,Z 493.427,A -85,B 0,C 180,E1 -27867.238,E2 -27867.238} C_VEL
LIN {X 0,Y 79.717,Z 484.99,A -85,B 0,C 180,E1 -27871.19,E2 -27871.19} C_VEL
LIN {X 0,Y 79.593,Z 484.194,A -85,B 0,C 180,E1 -27871.574,E2 -27871.574} C_VEL
LIN {X 0,Y 79.528,Z 484.204,A -85,B 0,C 180,E1 -27879.3,E2 -27879.3} C_VEL
LIN {X 0,Y 79.841,Z 484.158,A -85,B 0,C 180,E1 -27885.526,E2 -27885.526} C_VEL
LIN {X 0,Y 79.992,Z 484.145,A -85,B 0,C 180,E1 -27889.881,E2 -27889.881} C_VEL
LIN {X 0,Y 80.649,Z 484.059,A -85,B 0,C 180,E1 -27900.001,E2 -27900.001} C_VEL
LIN {X 0,Y 79.993,Z 484.137,A -85,B 0,C 180,E1 -27910.121,E2 -27910.121} C_VEL
LIN {X 0,Y 79.762,Z 484.174,A -85,B 0,C 180,E1 -27915.329,E2 -27915.329} C_VEL
LIN {X 0,Y 79.513,Z 484.198,A -85,B 0,C 180,E1 -27920.706,E2 -27920.706} C_VEL
LIN {X 0,Y 79.483,Z 484.201,A -85,B 0,C 180,E1 -27927.847,E2 -27927.847} C_VEL
LIN {X 0,Y 79.384,Z 484.222,A -85,B 0,C 180,E1 -27932.087,E2 -27932.087} C_VEL
LIN {X 0,Y 79.373,Z 484.216,A -85,B 0,C 180,E1 -27938.303,E2 -27938.303} C_VEL
LIN {X 0,Y 79.411,Z 484.21,A -85,B 0,C 180,E1 -27945.075,E2 -27945.075} C_VEL
LIN {X 0,Y 79.395,Z 484.216,A -85,B 0,C 180,E1 -27952.816,E2 -27952.816} C_VEL
LIN {X 0,Y 79.386,Z 484.22,A -85,B 0,C 180,E1 -27957.916,E2 -27957.916} C_VEL
LIN {X 0,Y 79.528,Z 484.195,A -85,B 0,C 180,E1 -27963.778,E2 -27963.778} C_VEL
LIN {X 0,Y 79.515,Z 484.204,A -85,B 0,C 180,E1 -27969.296,E2 -27969.296} C_VEL
LIN {X 0,Y 79.827,Z 484.166,A -85,B 0,C 180,E1 -27975.573,E2 -27975.573} C_VEL
LIN {X 0,Y 79.969,Z 484.142,A -85,B 0,C 180,E1 -27979.877,E2 -27979.877} C_VEL
LIN {X 0,Y 80.611,Z 484.059,A -85,B 0,C 180,E1 -27989.779,E2 -27989.779} C_VEL
LIN {X 0,Y 80.725,Z 484.461,A -85,B 0,C 180,E1 -27992.456,E2 -27992.456} C_VEL
LIN {X 0,Y 80.107,Z 486.343,A -85,B 0,C 180,E1 -27996.308,E2 -27996.308} C_VEL
LIN {X 0,Y 79.131,Z 489.288,A -85,B 0,C 180,E1 -27999.877,E2 -27999.877} C_VEL
LIN {X 0,Y 78.144,Z 494.521,A -85,B 0,C 180,E1 -28004.332,E2 -28004.332} C_VEL
LIN {X 0,Y 78.435,Z 499.059,A -85,B 0,C 180,E1 -28007.231,E2 -28007.231} C_VEL
LIN {X 0,Y 78.851,Z 500.653,A -85,B 0,C 180,E1 -28008.071,E2 -28008.071} C_VEL
LIN {X 0,Y 82.208,Z 511.746,A -85,B 0,C 180,E1 -28013.576,E2 -28013.576} C_VEL
LIN {X 0,Y 84.741,Z 523.186,A -85,B 0,C 180,E1 -28019.159,E2 -28019.159} C_VEL
LIN {X 0,Y 85.481,Z 526.71,A -85,B 0,C 180,E1 -28020.92,E2 -28020.92} C_VEL
LIN {X 0,Y 80.923,Z 539.06,A -85,B 0,C 180,E1 -28026.548,E2 -28026.548} C_VEL
LIN {X 0,Y 76.889,Z 549.925,A -85,B 0,C 180,E1 -28033.008,E2 -28033.008} C_VEL
LIN {X 0,Y 73.357,Z 561.008,A -85,B 0,C 180,E1 -28041.61,E2 -28041.61} C_VEL
LIN {X 0,Y 71.523,Z 568.433,A -85,B 0,C 180,E1 -28048.943,E2 -28048.943} C_VEL
LIN {X 0,Y 70.376,Z 575.994,A -85,B 0,C 180,E1 -28058.006,E2 -28058.006} C_VEL
LIN {X 0,Y 70.567,Z 583.179,A -85,B 0,C 180,E1 -28068.509,E2 -28068.509} C_VEL
LIN {X 0,Y 73.129,Z 589.693,A -85,B 0,C 180,E1 -28079.999,E2 -28079.999} C_VEL
LIN {X 0,Y 78.919,Z 595.445,A -85,B 0,C 180,E1 -28091.602,E2 -28091.602} C_VEL
LIN {X 0,Y 85.26,Z 598.872,A -85,B 0,C 180,E1 -28099.251,E2 -28099.251} C_VEL
LIN {X 0,Y 94.368,Z 601.852,A -85,B 0,C 180,E1 -28106.541,E2 -28106.541} C_VEL
LIN {X 0,Y 106.349,Z 604.044,A -85,B 0,C 180,E1 -28113.144,E2 -28113.144} C_VEL
LIN {X 0,Y 105.236,Z 604.197,A -85,B 0,C 180,E1 -28114.806,E2 -28114.806} C_VEL
LIN {X 0,Y 93.62,Z 603.606,A -85,B 0,C 180,E1 -28121.351,E2 -28121.351} C_VEL
LIN {X 0,Y 84.922,Z 602.222,A -85,B 0,C 180,E1 -28128.543,E2 -28128.543} C_VEL
LIN {X 0,Y 78.215,Z 599.984,A -85,B 0,C 180,E1 -28137.376,E2 -28137.376} C_VEL
LIN {X 0,Y 73.894,Z 596.845,A -85,B 0,C 180,E1 -28147.64,E2 -28147.64} C_VEL
LIN {X 0,Y 72.351,Z 592.734,A -85,B 0,C 180,E1 -28158.798,E2 -28158.798} C_VEL
LIN {X 0,Y 72.461,Z 590.176,A -85,B 0,C 180,E1 -28164.434,E2 -28164.434} C_VEL
LIN {X 0,Y 72.416,Z 587.037,A -85,B 0,C 180,E1 -28170,E2 -28170} C_VEL
LIN {X 0,Y 72.274,Z 581.047,A -85,B 0,C 180,E1 -28178.387,E2 -28178.387} C_VEL
LIN {X 0,Y 73.171,Z 573.719,A -85,B 0,C 180,E1 -28186.747,E2 -28186.747} C_VEL
LIN {X 0,Y 75.913,Z 563.411,A -85,B 0,C 180,E1 -28196.088,E2 -28196.088} C_VEL
LIN {X 0,Y 78.924,Z 554.58,A -85,B 0,C 180,E1 -28202.295,E2 -28202.295} C_VEL
LIN {X 0,Y 81.02,Z 548.534,A -85,B 0,C 180,E1 -28205.839,E2 -28205.839} C_VEL
LIN {X 0,Y 81.24,Z 536.098,A -85,B 0,C 180,E1 -28212.338,E2 -28212.338} C_VEL
LIN {X 0,Y 81.489,Z 523.165,A -85,B 0,C 180,E1 -28218.035,E2 -28218.035} C_VEL
LIN {X 0,Y 81.647,Z 512.322,A -85,B 0,C 180,E1 -28222.172,E2 -28222.172} C_VEL
LIN {X 0,Y 80.555,Z 506.202,A -85,B 0,C 180,E1 -28224.657,E2 -28224.657} C_VEL
LIN {X 0,Y 77.913,Z 496.647,A -85,B 0,C 180,E1 -28228.758,E2 -28228.758} C_VEL
LIN {X 0,Y 73.861,Z 488.402,A -85,B 0,C 180,E1 -28233.131,E2 -28233.131} C_VEL
LIN {X 0,Y 72.518,Z 485.382,A -85,B 0,C 180,E1 -28234.722,E2 -28234.722} C_VEL
LIN {X 0,Y 72.455,Z 485.071,A -85,B 0,C 180,E1 -28234.89,E2 -28234.89} C_VEL
LIN {X 0,Y 72.756,Z 485.039,A -85,B 0,C 180,E1 -28245.005,E2 -28245.005} C_VEL
LIN {X 0,Y 72.879,Z 485.032,A -85,B 0,C 180,E1 -28248.881,E2 -28248.881} C_VEL
LIN {X 0,Y 73.576,Z 484.94,A -85,B 0,C 180,E1 -28260.001,E2 -28260.001} C_VEL
LIN {X 0,Y 72.879,Z 485.023,A -85,B 0,C 180,E1 -28271.121,E2 -28271.121} C_VEL
LIN {X 0,Y 72.582,Z 485.066,A -85,B 0,C 180,E1 -28276.888,E2 -28276.888} C_VEL
LIN {X 0,Y 72.394,Z 485.092,A -85,B 0,C 180,E1 -28282.851,E2 -28282.851} C_VEL
LIN {X 0,Y 72.377,Z 485.086,A -85,B 0,C 180,E1 -28289.084,E2 -28289.084} C_VEL
LIN {X 0,Y 72.3,Z 485.097,A -85,B 0,C 180,E1 -28295.68,E2 -28295.68} C_VEL
LIN {X 0,Y 72.263,Z 485.107,A -85,B 0,C 180,E1 -28302.907,E2 -28302.907} C_VEL
LIN {X 0,Y 72.302,Z 485.103,A -85,B 0,C 180,E1 -28311.046,E2 -28311.046} C_VEL
LIN {X 0,Y 72.302,Z 485.094,A -85,B 0,C 180,E1 -28314.323,E2 -28314.323} C_VEL
LIN {X 0,Y 72.394,Z 485.09,A -85,B 0,C 180,E1 -28320.962,E2 -28320.962} C_VEL
LIN {X 0,Y 72.396,Z 485.092,A -85,B 0,C 180,E1 -28327.151,E2 -28327.151} C_VEL
LIN {X 0,Y 72.724,Z 485.049,A -85,B 0,C 180,E1 -28335.11,E2 -28335.11} C_VEL
LIN {X 0,Y 72.86,Z 485.03,A -85,B 0,C 180,E1 -28338.877,E2 -28338.877} C_VEL
LIN {X 0,Y 73.573,Z 484.936,A -85,B 0,C 180,E1 -28350,E2 -28350} C_VEL
LIN {X 0,Y 72.918,Z 485.014,A -85,B 0,C 180,E1 -28359.885,E2 -28359.885} C_VEL
LIN {X 0,Y 73.566,Z 487.298,A -85,B 0,C 180,E1 -28361.015,E2 -28361.015} C_VEL
LIN {X 0,Y 76.757,Z 494.882,A -85,B 0,C 180,E1 -28365.12,E2 -28365.12} C_VEL
LIN {X 0,Y 78.851,Z 500.653,A -85,B 0,C 180,E1 -28368.071,E2 -28368.071} C_VEL
LIN {X 0,Y 79.997,Z 505.592,A -85,B 0,C 180,E1 -28370.375,E2 -28370.375} C_VEL
LIN {X 0,Y 80.441,Z 510.724,A -85,B 0,C 180,E1 -28372.575,E2 -28372.575} C_VEL
LIN {X 0,Y 80.136,Z 517.672,A -85,B 0,C 180,E1 -28375.449,E2 -28375.449} C_VEL
LIN {X 0,Y 79.66,Z 521.132,A -85,B 0,C 180,E1 -28376.899,E2 -28376.899} C_VEL
LIN {X 0,Y 78.182,Z 527.903,A -85,B 0,C 180,E1 -28379.906,E2 -28379.906} C_VEL
LIN {X 0,Y 73.76,Z 539.488,A -85,B 0,C 180,E1 -28385.65,E2 -28385.65} C_VEL
LIN {X 0,Y 69.515,Z 550.458,A -85,B 0,C 180,E1 -28392.861,E2 -28392.861} C_VEL
LIN {X 0,Y 66.01,Z 561.214,A -85,B 0,C 180,E1 -28402.25,E2 -28402.25} C_VEL
LIN {X 0,Y 64.099,Z 569.361,A -85,B 0,C 180,E1 -28411.297,E2 -28411.297} C_VEL
LIN {X 0,Y 63.297,Z 576.225,A -85,B 0,C 180,E1 -28420.542,E2 -28420.542} C_VEL
LIN {X 0,Y 63.956,Z 582.899,A -85,B 0,C 180,E1 -28431.487,E2 -28431.487} C_VEL
LIN {X 0,Y 66.917,Z 589.066,A -85,B 0,C 180,E1 -28443.009,E2 -28443.009} C_VEL
LIN {X 0,Y 72.256,Z 594.131,A -85,B 0,C 180,E1 -28453.435,E2 -28453.435} C_VEL
LIN {X 0,Y 78.401,Z 597.703,A -85,B 0,C 180,E1 -28461.011,E2 -28461.011} C_VEL
LIN {X 0,Y 88.507,Z 601.328,A -85,B 0,C 180,E1 -28469.138,E2 -28469.138} C_VEL
LIN {X 0,Y 95.829,Z 603.087,A -85,B 0,C 180,E1 -28473.357,E2 -28473.357} C_VEL
LIN {X 0,Y 95.189,Z 603.141,A -85,B 0,C 180,E1 -28474.425,E2 -28474.425} C_VEL
LIN {X 0,Y 81.605,Z 601.275,A -85,B 0,C 180,E1 -28483.548,E2 -28483.548} C_VEL
LIN {X 0,Y 72.45,Z 598.377,A -85,B 0,C 180,E1 -28494.407,E2 -28494.407} C_VEL
LIN {X 0,Y 67.572,Z 595,A -85,B 0,C 180,E1 -28505.416,E2 -28505.416} C_VEL
LIN {X 0,Y 65.687,Z 590.636,A -85,B 0,C 180,E1 -28517.644,E2 -28517.644} C_VEL
LIN {X 0,Y 65.77,Z 587.956,A -85,B 0,C 180,E1 -28523.866,E2 -28523.866} C_VEL
LIN {X 0,Y 65.764,Z 586.416,A -85,B 0,C 180,E1 -28526.937,E2 -28526.937} C_VEL
LIN {X 0,Y 65.42,Z 580.557,A -85,B 0,C 180,E1 -28536.167,E2 -28536.167} C_VEL
LIN {X 0,Y 66.034,Z 573.538,A -85,B 0,C 180,E1 -28545.242,E2 -28545.242} C_VEL
LIN {X 0,Y 68.154,Z 564.753,A -85,B 0,C 180,E1 -28554.36,E2 -28554.36} C_VEL
LIN {X 0,Y 71.702,Z 554.406,A -85,B 0,C 180,E1 -28562.621,E2 -28562.621} C_VEL
LIN {X 0,Y 73.95,Z 548.47,A -85,B 0,C 180,E1 -28566.439,E2 -28566.439} C_VEL
LIN {X 0,Y 74.296,Z 536.587,A -85,B 0,C 180,E1 -28573.299,E2 -28573.299} C_VEL
LIN {X 0,Y 74.722,Z 523.804,A -85,B 0,C 180,E1 -28579.56,E2 -28579.56} C_VEL
LIN {X 0,Y 75.022,Z 513.089,A -85,B 0,C 180,E1 -28584.071,E2 -28584.071} C_VEL
LIN {X 0,Y 72.653,Z 501.987,A -85,B 0,C 180,E1 -28589.279,E2 -28589.279} C_VEL
LIN {X 0,Y 70.666,Z 497.207,A -85,B 0,C 180,E1 -28591.92,E2 -28591.92} C_VEL
LIN {X 0,Y 66.839,Z 489.473,A -85,B 0,C 180,E1 -28596.778,E2 -28596.778} C_VEL
LIN {X 0,Y 65.441,Z 486.515,A -85,B 0,C 180,E1 -28598.75,E2 -28598.75} C_VEL
LIN {X 0,Y 65.352,Z 485.969,A -85,B 0,C 180,E1 -28599.132,E2 -28599.132} C_VEL
LIN {X 0,Y 65.651,Z 485.923,A -85,B 0,C 180,E1 -28604.461,E2 -28604.461} C_VEL
LIN {X 0,Y 65.779,Z 485.916,A -85,B 0,C 180,E1 -28607.663,E2 -28607.663} C_VEL
LIN {X 0,Y 66.5,Z 485.821,A -85,B 0,C 180,E1 -28620.001,E2 -28620.001} C_VEL
LIN {X 0,Y 65.772,Z 485.911,A -85,B 0,C 180,E1 -28632.341,E2 -28632.341} C_VEL
LIN {X 0,Y 65.384,Z 485.956,A -85,B 0,C 180,E1 -28638.813,E2 -28638.813} C_VEL
LIN {X 0,Y 65.239,Z 485.981,A -85,B 0,C 180,E1 -28645.527,E2 -28645.527} C_VEL
LIN {X 0,Y 65.198,Z 485.989,A -85,B 0,C 180,E1 -28652.615,E2 -28652.615} C_VEL
LIN {X 0,Y 65.195,Z 485.989,A -85,B 0,C 180,E1 -28661.011,E2 -28661.011} C_VEL
LIN {X 0,Y 65.213,Z 485.987,A -85,B 0,C 180,E1 -28669.714,E2 -28669.714} C_VEL
LIN {X 0,Y 65.256,Z 485.982,A -85,B 0,C 180,E1 -28679.498,E2 -28679.498} C_VEL
LIN {X 0,Y 65.247,Z 485.974,A -85,B 0,C 180,E1 -28684.479,E2 -28684.479} C_VEL
LIN {X 0,Y 65.627,Z 485.931,A -85,B 0,C 180,E1 -28694.543,E2 -28694.543} C_VEL
LIN {X 0,Y 65.757,Z 485.918,A -85,B 0,C 180,E1 -28697.658,E2 -28697.658} C_VEL
LIN {X 0,Y 66.496,Z 485.817,A -85,B 0,C 180,E1 -28710,E2 -28710} C_VEL
LIN {X 0,Y 65.97,Z 485.979,A -85,B 0,C 180,E1 -28715.924,E2 -28715.924} C_VEL
LIN {X 0,Y 66.828,Z 488.637,A -85,B 0,C 180,E1 -28717.554,E2 -28717.554} C_VEL
LIN {X 0,Y 69.612,Z 494.829,A -85,B 0,C 180,E1 -28721.649,E2 -28721.649} C_VEL
LIN {X 0,Y 73.117,Z 504.992,A -85,B 0,C 180,E1 -28727.48,E2 -28727.48} C_VEL
LIN {X 0,Y 76.009,Z 515.438,A -85,B 0,C 180,E1 -28733.139,E2 -28733.139} C_VEL
LIN {X 0,Y 78.392,Z 527.128,A -85,B 0,C 180,E1 -28739.543,E2 -28739.543} C_VEL
LIN {X 0,Y 78.182,Z 527.903,A -85,B 0,C 180,E1 -28739.906,E2 -28739.906} C_VEL
LIN {X 0,Y 76.955,Z 531.117,A -85,B 0,C 180,E1 -28741.344,E2 -28741.344} C_VEL
LIN {X 0,Y 74.104,Z 535.59,A -85,B 0,C 180,E1 -28743.301,E2 -28743.301} C_VEL
LIN {X 0,Y 64.718,Z 546.403,A -85,B 0,C 180,E1 -28749.224,E2 -28749.224} C_VEL
LIN {X 0,Y 62.227,Z 550.53,A -85,B 0,C 180,E1 -28752.44,E2 -28752.44} C_VEL
LIN {X 0,Y 58.674,Z 561.562,A -85,B 0,C 180,E1 -28763.207,E2 -28763.207} C_VEL
LIN {X 0,Y 56.78,Z 570.249,A -85,B 0,C 180,E1 -28774.327,E2 -28774.327} C_VEL
LIN {X 0,Y 56.499,Z 577.383,A -85,B 0,C 180,E1 -28785.593,E2 -28785.593} C_VEL
LIN {X 0,Y 58.697,Z 585.097,A -85,B 0,C 180,E1 -28799.999,E2 -28799.999} C_VEL
LIN {X 0,Y 63.903,Z 591.254,A -85,B 0,C 180,E1 -28812.705,E2 -28812.705} C_VEL
LIN {X 0,Y 71.665,Z 596.243,A -85,B 0,C 180,E1 -28823.095,E2 -28823.095} C_VEL
LIN {X 0,Y 83.014,Z 600.64,A -85,B 0,C 180,E1 -28832.158,E2 -28832.158} C_VEL
LIN {X 0,Y 84.982,Z 601.297,A -85,B 0,C 180,E1 -28834.21,E2 -28834.21} C_VEL
LIN {X 0,Y 75.012,Z 599.369,A -85,B 0,C 180,E1 -28841.451,E2 -28841.451} C_VEL
LIN {X 0,Y 66.954,Z 596.633,A -85,B 0,C 180,E1 -28850.965,E2 -28850.965} C_VEL
LIN {X 0,Y 60.516,Z 591.987,A -85,B 0,C 180,E1 -28866.017,E2 -28866.017} C_VEL
LIN {X 0,Y 59.016,Z 587.055,A -85,B 0,C 180,E1 -28879.71,E2 -28879.71} C_VEL
LIN {X 0,Y 59.097,Z 585.659,A -85,B 0,C 180,E1 -28883.17,E2 -28883.17} C_VEL
LIN {X 0,Y 59.003,Z 583.982,A -85,B 0,C 180,E1 -28886.586,E2 -28886.586} C_VEL
LIN {X 0,Y 58.591,Z 577.788,A -85,B 0,C 180,E1 -28896.889,E2 -28896.889} C_VEL
LIN {X 0,Y 59.403,Z 570.089,A -85,B 0,C 180,E1 -28907.334,E2 -28907.334} C_VEL
LIN {X 0,Y 61.929,Z 561.181,A -85,B 0,C 180,E1 -28916.996,E2 -28916.996} C_VEL
LIN {X 0,Y 65.961,Z 550.345,A -85,B 0,C 180,E1 -28925.874,E2 -28925.874} C_VEL
LIN {X 0,Y 66.791,Z 548.329,A -85,B 0,C 180,E1 -28927.231,E2 -28927.231} C_VEL
LIN {X 0,Y 67.296,Z 538.626,A -85,B 0,C 180,E1 -28933.506,E2 -28933.506} C_VEL
LIN {X 0,Y 67.907,Z 526.659,A -85,B 0,C 180,E1 -28940.153,E2 -28940.153} C_VEL
LIN {X 0,Y 68.472,Z 515.137,A -85,B 0,C 180,E1 -28945.629,E2 -28945.629} C_VEL
LIN {X 0,Y 66.909,Z 506.679,A -85,B 0,C 180,E1 -28950.072,E2 -28950.072} C_VEL
LIN {X 0,Y 65.88,Z 502.954,A -85,B 0,C 180,E1 -28952.179,E2 -28952.179} C_VEL
LIN {X 0,Y 61.874,Z 494.26,A -85,B 0,C 180,E1 -28958.338,E2 -28958.338} C_VEL
LIN {X 0,Y 60.28,Z 490.872,A -85,B 0,C 180,E1 -28960.949,E2 -28960.949} C_VEL
LIN {X 0,Y 58.743,Z 488.063,A -85,B 0,C 180,E1 -28963.319,E2 -28963.319} C_VEL
LIN {X 0,Y 58.555,Z 486.806,A -85,B 0,C 180,E1 -28964.161,E2 -28964.161} C_VEL
LIN {X 0,Y 58.817,Z 486.774,A -85,B 0,C 180,E1 -28973.139,E2 -28973.139} C_VEL
LIN {X 0,Y 59.392,Z 486.706,A -85,B 0,C 180,E1 -28980.001,E2 -28980.001} C_VEL
LIN {X 0,Y 58.817,Z 486.783,A -85,B 0,C 180,E1 -28986.864,E2 -28986.864} C_VEL
LIN {X 0,Y 58.525,Z 486.819,A -85,B 0,C 180,E1 -28996.124,E2 -28996.124} C_VEL
LIN {X 0,Y 58.15,Z 486.857,A -85,B 0,C 180,E1 -29008.912,E2 -29008.912} C_VEL
LIN {X 0,Y 58.159,Z 486.866,A -85,B 0,C 180,E1 -29012.235,E2 -29012.235} C_VEL
LIN {X 0,Y 58.038,Z 486.87,A -85,B 0,C 180,E1 -29017.264,E2 -29017.264} C_VEL
LIN {X 0,Y 58.023,Z 486.873,A -85,B 0,C 180,E1 -29026.617,E2 -29026.617} C_VEL
LIN {X 0,Y 58.039,Z 486.874,A -85,B 0,C 180,E1 -29032.739,E2 -29032.739} C_VEL
LIN {X 0,Y 58.161,Z 486.864,A -85,B 0,C 180,E1 -29037.768,E2 -29037.768} C_VEL
LIN {X 0,Y 58.154,Z 486.862,A -85,B 0,C 180,E1 -29041.093,E2 -29041.093} C_VEL
LIN {X 0,Y 58.519,Z 486.814,A -85,B 0,C 180,E1 -29053.907,E2 -29053.907} C_VEL
LIN {X 0,Y 58.801,Z 486.78,A -85,B 0,C 180,E1 -29063.136,E2 -29063.136} C_VEL
LIN {X 0,Y 59.304,Z 486.714,A -85,B 0,C 180,E1 -29070.849,E2 -29070.849} C_VEL
LIN {X 0,Y 59.398,Z 487.611,A -85,B 0,C 180,E1 -29071.695,E2 -29071.695} C_VEL
LIN {X 0,Y 63.879,Z 498.449,A -85,B 0,C 180,E1 -29079.819,E2 -29079.819} C_VEL
LIN {X 0,Y 67.19,Z 509.033,A -85,B 0,C 180,E1 -29086.717,E2 -29086.717} C_VEL
LIN {X 0,Y 69.517,Z 518.098,A -85,B 0,C 180,E1 -29092.278,E2 -29092.278} C_VEL
LIN {X 0,Y 71.374,Z 527.691,A -85,B 0,C 180,E1 -29098.044,E2 -29098.044} C_VEL
LIN {X 0,Y 67.365,Z 537.839,A -85,B 0,C 180,E1 -29103.422,E2 -29103.422} C_VEL
LIN {X 0,Y 62.564,Z 549.74,A -85,B 0,C 180,E1 -29111.77,E2 -29111.77} C_VEL
LIN {X 0,Y 62.227,Z 550.53,A -85,B 0,C 180,E1 -29112.44,E2 -29112.44} C_VEL
LIN {X 0,Y 59.99,Z 554.565,A -85,B 0,C 180,E1 -29115.971,E2 -29115.971} C_VEL
LIN {X 0,Y 55.142,Z 560.455,A -85,B 0,C 180,E1 -29122.269,E2 -29122.269} C_VEL
LIN {X 0,Y 51.591,Z 564.883,A -85,B 0,C 180,E1 -29128.326,E2 -29128.326} C_VEL
LIN {X 0,Y 49.985,Z 568.21,A -85,B 0,C 180,E1 -29133.613,E2 -29133.613} C_VEL
LIN {X 0,Y 49.771,Z 569.339,A -85,B 0,C 180,E1 -29135.478,E2 -29135.478} C_VEL
LIN {X 0,Y 49.911,Z 577.637,A -85,B 0,C 180,E1 -29150.283,E2 -29150.283} C_VEL
LIN {X 0,Y 52.591,Z 584.17,A -85,B 0,C 180,E1 -29163.83,E2 -29163.83} C_VEL
LIN {X 0,Y 59.109,Z 590.836,A -85,B 0,C 180,E1 -29177.979,E2 -29177.979} C_VEL
LIN {X 0,Y 69.964,Z 596.839,A -85,B 0,C 180,E1 -29190.148,E2 -29190.148} C_VEL
LIN {X 0,Y 73.958,Z 598.413,A -85,B 0,C 180,E1 -29193.12,E2 -29193.12} C_VEL
LIN {X 0,Y 73.382,Z 598.426,A -85,B 0,C 180,E1 -29195.073,E2 -29195.073} C_VEL
LIN {X 0,Y 61.757,Z 594.779,A -85,B 0,C 180,E1 -29206.937,E2 -29206.937} C_VEL
LIN {X 0,Y 54.299,Z 589.675,A -85,B 0,C 180,E1 -29223.479,E2 -29223.479} C_VEL
LIN {X 0,Y 52.467,Z 584.657,A -85,B 0,C 180,E1 -29238.409,E2 -29238.409} C_VEL
LIN {X 0,Y 52.491,Z 583.134,A -85,B 0,C 180,E1 -29242.306,E2 -29242.306} C_VEL
LIN {X 0,Y 51.98,Z 579.351,A -85,B 0,C 180,E1 -29250,E2 -29250} C_VEL
LIN {X 0,Y 52.003,Z 572.394,A -85,B 0,C 180,E1 -29261.696,E2 -29261.696} C_VEL
LIN {X 0,Y 54.016,Z 562.783,A -85,B 0,C 180,E1 -29274.392,E2 -29274.392} C_VEL
LIN {X 0,Y 58.034,Z 551.891,A -85,B 0,C 180,E1 -29285.115,E2 -29285.115} C_VEL
LIN {X 0,Y 59.669,Z 547.927,A -85,B 0,C 180,E1 -29288.196,E2 -29288.196} C_VEL
LIN {X 0,Y 60.368,Z 538.275,A -85,B 0,C 180,E1 -29295.14,E2 -29295.14} C_VEL
LIN {X 0,Y 61.313,Z 524.862,A -85,B 0,C 180,E1 -29303.356,E2 -29303.356} C_VEL
LIN {X 0,Y 61.886,Z 517.324,A -85,B 0,C 180,E1 -29307.357,E2 -29307.357} C_VEL
LIN {X 0,Y 61.377,Z 512.849,A -85,B 0,C 180,E1 -29309.938,E2 -29309.938} C_VEL
LIN {X 0,Y 60.021,Z 506.501,A -85,B 0,C 180,E1 -29313.955,E2 -29313.955} C_VEL
LIN {X 0,Y 56.226,Z 497.75,A -85,B 0,C 180,E1 -29321.04,E2 -29321.04} C_VEL
LIN {X 0,Y 53.46,Z 491.626,A -85,B 0,C 180,E1 -29326.701,E2 -29326.701} C_VEL
LIN {X 0,Y 52.495,Z 490.36,A -85,B 0,C 180,E1 -29328.417,E2 -29328.417} C_VEL
LIN {X 0,Y 51.651,Z 487.669,A -85,B 0,C 180,E1 -29331.196,E2 -29331.196} C_VEL
LIN {X 0,Y 52.276,Z 487.591,A -85,B 0,C 180,E1 -29340.002,E2 -29340.002} C_VEL
LIN {X 0,Y 51.692,Z 487.668,A -85,B 0,C 180,E1 -29347.816,E2 -29347.816} C_VEL
LIN {X 0,Y 51.393,Z 487.704,A -85,B 0,C 180,E1 -29356.818,E2 -29356.818} C_VEL
LIN {X 0,Y 51.024,Z 487.754,A -85,B 0,C 180,E1 -29364.409,E2 -29364.409} C_VEL
LIN {X 0,Y 51.032,Z 487.75,A -85,B 0,C 180,E1 -29374.281,E2 -29374.281} C_VEL
LIN {X 0,Y 50.989,Z 487.749,A -85,B 0,C 180,E1 -29386.437,E2 -29386.437} C_VEL
LIN {X 0,Y 51.054,Z 487.744,A -85,B 0,C 180,E1 -29396.59,E2 -29396.59} C_VEL
LIN {X 0,Y 51.027,Z 487.748,A -85,B 0,C 180,E1 -29405.595,E2 -29405.595} C_VEL
LIN {X 0,Y 51.46,Z 487.693,A -85,B 0,C 180,E1 -29414.149,E2 -29414.149} C_VEL
LIN {X 0,Y 51.795,Z 487.733,A -85,B 0,C 180,E1 -29423.915,E2 -29423.915} C_VEL
LIN {X 0,Y 52.585,Z 489.926,A -85,B 0,C 180,E1 -29426.168,E2 -29426.168} C_VEL
LIN {X 0,Y 53.67,Z 491.279,A -85,B 0,C 180,E1 -29428.124,E2 -29428.124} C_VEL
LIN {X 0,Y 55.478,Z 495.062,A -85,B 0,C 180,E1 -29431.996,E2 -29431.996} C_VEL
LIN {X 0,Y 58.446,Z 503.023,A -85,B 0,C 180,E1 -29438.645,E2 -29438.645} C_VEL
LIN {X 0,Y 60.951,Z 511.818,A -85,B 0,C 180,E1 -29445.036,E2 -29445.036} C_VEL
LIN {X 0,Y 63.132,Z 521.312,A -85,B 0,C 180,E1 -29451.638,E2 -29451.638} C_VEL
LIN {X 0,Y 64.386,Z 528.361,A -85,B 0,C 180,E1 -29456.453,E2 -29456.453} C_VEL
LIN {X 0,Y 59.184,Z 540.586,A -85,B 0,C 180,E1 -29463.771,E2 -29463.771} C_VEL
LIN {X 0,Y 54.753,Z 551.143,A -85,B 0,C 180,E1 -29472.431,E2 -29472.431} C_VEL
LIN {X 0,Y 51.298,Z 561.894,A -85,B 0,C 180,E1 -29484.631,E2 -29484.631} C_VEL
LIN {X 0,Y 49.771,Z 569.339,A -85,B 0,C 180,E1 -29495.478,E2 -29495.478} C_VEL
LIN {X 0,Y 48.92,Z 572.544,A -85,B 0,C 180,E1 -29501.18,E2 -29501.18} C_VEL
LIN {X 0,Y 47.538,Z 575.282,A -85,B 0,C 180,E1 -29507.229,E2 -29507.229} C_VEL
LIN {X 0,Y 45.789,Z 580.935,A -85,B 0,C 180,E1 -29522.851,E2 -29522.851} C_VEL
LIN {X 0,Y 47.056,Z 583.469,A -85,B 0,C 180,E1 -29529.34,E2 -29529.34} C_VEL
LIN {X 0,Y 54.066,Z 589.688,A -85,B 0,C 180,E1 -29542.951,E2 -29542.951} C_VEL
LIN {X 0,Y 63.82,Z 595.087,A -85,B 0,C 180,E1 -29553.408,E2 -29553.408} C_VEL
LIN {X 0,Y 61.568,Z 594.485,A -85,B 0,C 180,E1 -29556.961,E2 -29556.961} C_VEL
LIN {X 0,Y 51.262,Z 589.796,A -85,B 0,C 180,E1 -29571.907,E2 -29571.907} C_VEL
LIN {X 0,Y 46.238,Z 583.589,A -85,B 0,C 180,E1 -29592.303,E2 -29592.303} C_VEL
LIN {X 0,Y 45.89,Z 580.513,A -85,B 0,C 180,E1 -29601.191,E2 -29601.191} C_VEL
LIN {X 0,Y 45.268,Z 576.475,A -85,B 0,C 180,E1 -29610,E2 -29610} C_VEL
LIN {X 0,Y 45.292,Z 569.074,A -85,B 0,C 180,E1 -29623.459,E2 -29623.459} C_VEL
LIN {X 0,Y 47.878,Z 559.065,A -85,B 0,C 180,E1 -29637.77,E2 -29637.77} C_VEL
LIN {X 0,Y 52.118,Z 548.483,A -85,B 0,C 180,E1 -29648.584,E2 -29648.584} C_VEL
LIN {X 0,Y 52.858,Z 546.357,A -85,B 0,C 180,E1 -29650.404,E2 -29650.404} C_VEL
LIN {X 0,Y 53.684,Z 535.391,A -85,B 0,C 180,E1 -29659.115,E2 -29659.115} C_VEL
LIN {X 0,Y 55.049,Z 522.424,A -85,B 0,C 180,E1 -29667.684,E2 -29667.684} C_VEL
LIN {X 0,Y 55.394,Z 517.258,A -85,B 0,C 180,E1 -29670.787,E2 -29670.787} C_VEL
LIN {X 0,Y 54.395,Z 510.65,A -85,B 0,C 180,E1 -29675.375,E2 -29675.375} C_VEL
LIN {X 0,Y 50.723,Z 501.417,A -85,B 0,C 180,E1 -29683.914,E2 -29683.914} C_VEL
LIN {X 0,Y 48.605,Z 496.278,A -85,B 0,C 180,E1 -29689.589,E2 -29689.589} C_VEL
LIN {X 0,Y 47.186,Z 493.111,A -85,B 0,C 180,E1 -29693.588,E2 -29693.588} C_VEL
LIN {X 0,Y 45.59,Z 490.671,A -85,B 0,C 180,E1 -29697.793,E2 -29697.793} C_VEL
LIN {X 0,Y 45.141,Z 488.479,A -85,B 0,C 180,E1 -29700.281,E2 -29700.281} C_VEL
LIN {X 0,Y 44.543,Z 488.553,A -85,B 0,C 180,E1 -29709.08,E2 -29709.08} C_VEL
LIN {X 0,Y 44.156,Z 488.6,A -85,B 0,C 180,E1 -29718.564,E2 -29718.564} C_VEL
LIN {X 0,Y 43.844,Z 488.638,A -85,B 0,C 180,E1 -29728.745,E2 -29728.745} C_VEL
LIN {X 0,Y 43.807,Z 488.649,A -85,B 0,C 180,E1 -29739.923,E2 -29739.923} C_VEL
LIN {X 0,Y 43.846,Z 488.639,A -85,B 0,C 180,E1 -29753.271,E2 -29753.271} C_VEL
LIN {X 0,Y 43.846,Z 488.642,A -85,B 0,C 180,E1 -29761.259,E2 -29761.259} C_VEL
LIN {X 0,Y 44.292,Z 488.609,A -85,B 0,C 180,E1 -29772.946,E2 -29772.946} C_VEL
LIN {X 0,Y 45.122,Z 490.964,A -85,B 0,C 180,E1 -29776.49,E2 -29776.49} C_VEL
LIN {X 0,Y 47.197,Z 493.24,A -85,B 0,C 180,E1 -29781.437,E2 -29781.437} C_VEL
LIN {X 0,Y 49.284,Z 496.808,A -85,B 0,C 180,E1 -29786.599,E2 -29786.599} C_VEL
LIN {X 0,Y 52.234,Z 505.011,A -85,B 0,C 180,E1 -29795.071,E2 -29795.071} C_VEL
LIN {X 0,Y 54.771,Z 514.896,A -85,B 0,C 180,E1 -29803.448,E2 -29803.448} C_VEL
LIN {X 0,Y 56.745,Z 524.418,A -85,B 0,C 180,E1 -29810.915,E2 -29810.915} C_VEL
LIN {X 0,Y 57.323,Z 528.238,A -85,B 0,C 180,E1 -29813.832,E2 -29813.832} C_VEL
LIN {X 0,Y 56.748,Z 530.465,A -85,B 0,C 180,E1 -29815.272,E2 -29815.272} C_VEL
LIN {X 0,Y 50.95,Z 543.037,A -85,B 0,C 180,E1 -29824.141,E2 -29824.141} C_VEL
LIN {X 0,Y 46.011,Z 555.03,A -85,B 0,C 180,E1 -29836.576,E2 -29836.576} C_VEL
LIN {X 0,Y 43.608,Z 563.405,A -85,B 0,C 180,E1 -29848.507,E2 -29848.507} C_VEL
LIN {X 0,Y 42.708,Z 570.334,A -85,B 0,C 180,E1 -29860.783,E2 -29860.783} C_VEL
LIN {X 0,Y 43.986,Z 578.312,A -85,B 0,C 180,E1 -29877.709,E2 -29877.709} C_VEL
LIN {X 0,Y 47.056,Z 583.469,A -85,B 0,C 180,E1 -29889.34,E2 -29889.34} C_VEL
LIN {X 0,Y 48.006,Z 585.049,A -85,B 0,C 180,E1 -29893.599,E2 -29893.599} C_VEL
LIN {X 0,Y 50.192,Z 588.777,A -85,B 0,C 180,E1 -29908.583,E2 -29908.583} C_VEL
LIN {X 0,Y 52.301,Z 590.131,A -85,B 0,C 180,E1 -29912.05,E2 -29912.05} C_VEL
LIN {X 0,Y 53.81,Z 590.953,A -85,B 0,C 180,E1 -29913.629,E2 -29913.629} C_VEL
LIN {X 0,Y 52.628,Z 590.607,A -85,B 0,C 180,E1 -29916.753,E2 -29916.753} C_VEL
LIN {X 0,Y 42.789,Z 584.992,A -85,B 0,C 180,E1 -29935.206,E2 -29935.206} C_VEL
LIN {X 0,Y 39.641,Z 579.41,A -85,B 0,C 180,E1 -29954.578,E2 -29954.578} C_VEL
LIN {X 0,Y 39.126,Z 576.756,A -85,B 0,C 180,E1 -29962.258,E2 -29962.258} C_VEL
LIN {X 0,Y 38.287,Z 570.977,A -85,B 0,C 180,E1 -29975.266,E2 -29975.266} C_VEL
LIN {X 0,Y 39.697,Z 561.385,A -85,B 0,C 180,E1 -29992.949,E2 -29992.949} C_VEL
LIN {X 0,Y 43.683,Z 551.029,A -85,B 0,C 180,E1 -30006.822,E2 -30006.822} C_VEL
LIN {X 0,Y 45.872,Z 545.834,A -85,B 0,C 180,E1 -30012.089,E2 -30012.089} C_VEL
LIN {X 0,Y 46.865,Z 535.763,A -85,B 0,C 180,E1 -30021.237,E2 -30021.237} C_VEL
LIN {X 0,Y 48.625,Z 522.696,A -85,B 0,C 180,E1 -30031.053,E2 -30031.053} C_VEL
LIN {X 0,Y 48.978,Z 519.081,A -85,B 0,C 180,E1 -30033.474,E2 -30033.474} C_VEL
LIN {X 0,Y 48.101,Z 512.995,A -85,B 0,C 180,E1 -30038.577,E2 -30038.577} C_VEL
LIN {X 0,Y 44.975,Z 503.994,A -85,B 0,C 180,E1 -30048.738,E2 -30048.738} C_VEL
LIN {X 0,Y 42.921,Z 498.858,A -85,B 0,C 180,E1 -30055.776,E2 -30055.776} C_VEL
LIN {X 0,Y 41.153,Z 494.943,A -85,B 0,C 180,E1 -30062.769,E2 -30062.769} C_VEL
LIN {X 0,Y 37.388,Z 491.21,A -85,B 0,C 180,E1 -30079.973,E2 -30079.973} C_VEL
LIN {X 0,Y 36.775,Z 489.519,A -85,B 0,C 180,E1 -30089.324,E2 -30089.324} C_VEL
LIN {X 0,Y 36.728,Z 489.53,A -85,B 0,C 180,E1 -30100.057,E2 -30100.057} C_VEL
LIN {X 0,Y 36.634,Z 489.684,A -85,B 0,C 180,E1 -30104.493,E2 -30104.493} C_VEL
LIN {X 0,Y 36.885,Z 490.332,A -85,B 0,C 180,E1 -30109.659,E2 -30109.659} C_VEL
LIN {X 0,Y 38.889,Z 493.748,A -85,B 0,C 180,E1 -30124.64,E2 -30124.64} C_VEL
LIN {X 0,Y 40.239,Z 494.646,A -85,B 0,C 180,E1 -30129.555,E2 -30129.555} C_VEL
LIN {X 0,Y 42.917,Z 498.762,A -85,B 0,C 180,E1 -30139.292,E2 -30139.292} C_VEL
LIN {X 0,Y 44.756,Z 502.522,A -85,B 0,C 180,E1 -30145.299,E2 -30145.299} C_VEL
LIN {X 0,Y 46.924,Z 509.995,A -85,B 0,C 180,E1 -30153.761,E2 -30153.761} C_VEL
LIN {X 0,Y 48.773,Z 518.975,A -85,B 0,C 180,E1 -30162.483,E2 -30162.483} C_VEL
LIN {X 0,Y 50.143,Z 526.581,A -85,B 0,C 180,E1 -30169.443,E2 -30169.443} C_VEL
LIN {X 0,Y 50.51,Z 529.325,A -85,B 0,C 180,E1 -30171.856,E2 -30171.856} C_VEL
LIN {X 0,Y 44.283,Z 542.068,A -85,B 0,C 180,E1 -30181.516,E2 -30181.516} C_VEL
LIN {X 0,Y 38.782,Z 554.741,A -85,B 0,C 180,E1 -30196.458,E2 -30196.458} C_VEL
LIN {X 0,Y 36.407,Z 563.298,A -85,B 0,C 180,E1 -30211.142,E2 -30211.142} C_VEL
LIN {X 0,Y 36.135,Z 571.409,A -85,B 0,C 180,E1 -30228.783,E2 -30228.783} C_VEL
LIN {X 0,Y 38.482,Z 578.176,A -85,B 0,C 180,E1 -30245.237,E2 -30245.237} C_VEL
LIN {X 0,Y 46.215,Z 586.201,A -85,B 0,C 180,E1 -30264.159,E2 -30264.159} C_VEL
LIN {X 0,Y 52.301,Z 590.131,A -85,B 0,C 180,E1 -30272.05,E2 -30272.05} C_VEL
LIN {X 0,Y 52.508,Z 590.339,A -85,B 0,C 180,E1 -30273.264,E2 -30273.264} C_VEL
LIN {X 0,Y 51.472,Z 590.003,A -85,B 0,C 180,E1 -30275.444,E2 -30275.444} C_VEL
LIN {X 0,Y 48.91,Z 588.868,A -85,B 0,C 180,E1 -30277.998,E2 -30277.998} C_VEL
LIN {X 0,Y 40.842,Z 584.555,A -85,B 0,C 180,E1 -30283.964,E2 -30283.964} C_VEL
LIN {X 0,Y 38.033,Z 582.736,A -85,B 0,C 180,E1 -30288.265,E2 -30288.265} C_VEL
LIN {X 0,Y 37.611,Z 582.412,A -85,B 0,C 180,E1 -30289.355,E2 -30289.355} C_VEL
LIN {X 0,Y 33.398,Z 576.58,A -85,B 0,C 180,E1 -30311.6,E2 -30311.6} C_VEL
LIN {X 0,Y 32.561,Z 573.675,A -85,B 0,C 180,E1 -30320.684,E2 -30320.684} C_VEL
LIN {X 0,Y 31.596,Z 567.587,A -85,B 0,C 180,E1 -30336.385,E2 -30336.385} C_VEL
LIN {X 0,Y 33.083,Z 558.781,A -85,B 0,C 180,E1 -30355.142,E2 -30355.142} C_VEL
LIN {X 0,Y 37.925,Z 547.511,A -85,B 0,C 180,E1 -30371.666,E2 -30371.666} C_VEL
LIN {X 0,Y 38.984,Z 544.98,A -85,B 0,C 180,E1 -30374.55,E2 -30374.55} C_VEL
LIN {X 0,Y 40.704,Z 532.554,A -85,B 0,C 180,E1 -30387.32,E2 -30387.32} C_VEL
LIN {X 0,Y 42.62,Z 521.618,A -85,B 0,C 180,E1 -30396.395,E2 -30396.395} C_VEL
LIN {X 0,Y 42.417,Z 517.103,A -85,B 0,C 180,E1 -30400.649,E2 -30400.649} C_VEL
LIN {X 0,Y 40.326,Z 509.786,A -85,B 0,C 180,E1 -30409.965,E2 -30409.965} C_VEL
LIN {X 0,Y 38.32,Z 503.454,A -85,B 0,C 180,E1 -30420.002,E2 -30420.002} C_VEL
LIN {X 0,Y 37.401,Z 500.807,A -85,B 0,C 180,E1 -30425.393,E2 -30425.393} C_VEL
LIN {X 0,Y 34.376,Z 497.228,A -85,B 0,C 180,E1 -30444.138,E2 -30444.138} C_VEL
LIN {X 0,Y 34.044,Z 496.088,A -85,B 0,C 180,E1 -30454.338,E2 -30454.338} C_VEL
LIN {X 0,Y 34.029,Z 496.085,A -85,B 0,C 180,E1 -30458.289,E2 -30458.289} C_VEL
LIN {X 0,Y 34.499,Z 498.225,A -85,B 0,C 180,E1 -30474.578,E2 -30474.578} C_VEL
LIN {X 0,Y 36.657,Z 500.713,A -85,B 0,C 180,E1 -30487.453,E2 -30487.453} C_VEL
LIN {X 0,Y 38.475,Z 504.008,A -85,B 0,C 180,E1 -30496.361,E2 -30496.361} C_VEL
LIN {X 0,Y 39.797,Z 507.15,A -85,B 0,C 180,E1 -30502.277,E2 -30502.277} C_VEL
LIN {X 0,Y 41.12,Z 512.935,A -85,B 0,C 180,E1 -30510,E2 -30510} C_VEL
LIN {X 0,Y 42.497,Z 521.338,A -85,B 0,C 180,E1 -30519.519,E2 -30519.519} C_VEL
LIN {X 0,Y 43.596,Z 528.806,A -85,B 0,C 180,E1 -30527.593,E2 -30527.593} C_VEL
LIN {X 0,Y 43.417,Z 530.209,A -85,B 0,C 180,E1 -30528.889,E2 -30528.889} C_VEL
LIN {X 0,Y 37.186,Z 542.094,A -85,B 0,C 180,E1 -30539.057,E2 -30539.057} C_VEL
LIN {X 0,Y 31.948,Z 553.218,A -85,B 0,C 180,E1 -30554.52,E2 -30554.52} C_VEL
LIN {X 0,Y 29.51,Z 561.629,A -85,B 0,C 180,E1 -30571.551,E2 -30571.551} C_VEL
LIN {X 0,Y 29.623,Z 569.989,A -85,B 0,C 180,E1 -30593.185,E2 -30593.185} C_VEL
LIN {X 0,Y 34.755,Z 578.838,A -85,B 0,C 180,E1 -30617.655,E2 -30617.655} C_VEL
LIN {X 0,Y 44.623,Z 586.506,A -85,B 0,C 180,E1 -30634.748,E2 -30634.748} C_VEL
LIN {X 0,Y 43.839,Z 586.169,A -85,B 0,C 180,E1 -30636.721,E2 -30636.721} C_VEL
LIN {X 0,Y 37.611,Z 582.412,A -85,B 0,C 180,E1 -30649.355,E2 -30649.355} C_VEL
LIN {X 0,Y 34.823,Z 580.085,A -85,B 0,C 180,E1 -30656.685,E2 -30656.685} C_VEL
LIN {X 0,Y 30.878,Z 576.061,A -85,B 0,C 180,E1 -30666.489,E2 -30666.489} C_VEL
LIN {X 0,Y 26.562,Z 570.137,A -85,B 0,C 180,E1 -30680.725,E2 -30680.725} C_VEL
LIN {X 0,Y 24.926,Z 565.093,A -85,B 0,C 180,E1 -30694.704,E2 -30694.704} C_VEL
LIN {X 0,Y 26.489,Z 556.274,A -85,B 0,C 180,E1 -30717.664,E2 -30717.664} C_VEL
LIN {X 0,Y 31.617,Z 545.589,A -85,B 0,C 180,E1 -30736.08,E2 -30736.08} C_VEL
LIN {X 0,Y 32.106,Z 544.618,A -85,B 0,C 180,E1 -30737.365,E2 -30737.365} C_VEL
LIN {X 0,Y 34.26,Z 532.716,A -85,B 0,C 180,E1 -30751.91,E2 -30751.91} C_VEL
LIN {X 0,Y 36.371,Z 523.415,A -85,B 0,C 180,E1 -30760.818,E2 -30760.818} C_VEL
LIN {X 0,Y 36.493,Z 520.16,A -85,B 0,C 180,E1 -30764.347,E2 -30764.347} C_VEL
LIN {X 0,Y 35.046,Z 513.445,A -85,B 0,C 180,E1 -30774.601,E2 -30774.601} C_VEL
LIN {X 0,Y 34.111,Z 508.967,A -85,B 0,C 180,E1 -30782.955,E2 -30782.955} C_VEL
LIN {X 0,Y 33.758,Z 507.657,A -85,B 0,C 180,E1 -30785.977,E2 -30785.977} C_VEL
LIN {X 0,Y 32.794,Z 505.871,A -85,B 0,C 180,E1 -30792.377,E2 -30792.377} C_VEL
LIN {X 0,Y 31.403,Z 503.525,A -85,B 0,C 180,E1 -30806.593,E2 -30806.593} C_VEL
LIN {X 0,Y 31.137,Z 503.27,A -85,B 0,C 180,E1 -30822.624,E2 -30822.624} C_VEL
LIN {X 0,Y 31.467,Z 504.756,A -85,B 0,C 180,E1 -30833.918,E2 -30833.918} C_VEL
LIN {X 0,Y 32.816,Z 506.582,A -85,B 0,C 180,E1 -30844.639,E2 -30844.639} C_VEL
LIN {X 0,Y 34.354,Z 509.887,A -85,B 0,C 180,E1 -30854.686,E2 -30854.686} C_VEL
LIN {X 0,Y 34.999,Z 512.671,A -85,B 0,C 180,E1 -30860.043,E2 -30860.043} C_VEL
LIN {X 0,Y 35.67,Z 517.686,A -85,B 0,C 180,E1 -30867.758,E2 -30867.758} C_VEL
LIN {X 0,Y 36.452,Z 525.529,A -85,B 0,C 180,E1 -30878.314,E2 -30878.314} C_VEL
LIN {X 0,Y 36.884,Z 529.593,A -85,B 0,C 180,E1 -30883.501,E2 -30883.501} C_VEL
LIN {X 0,Y 35.917,Z 531.965,A -85,B 0,C 180,E1 -30885.648,E2 -30885.648} C_VEL
LIN {X 0,Y 29.19,Z 543.658,A -85,B 0,C 180,E1 -30897.915,E2 -30897.915} C_VEL
LIN {X 0,Y 23.993,Z 554.841,A -85,B 0,C 180,E1 -30918.766,E2 -30918.766} C_VEL
LIN {X 0,Y 22.42,Z 562.88,A -85,B 0,C 180,E1 -30941.728,E2 -30941.728} C_VEL
LIN {X 0,Y 24.636,Z 570.772,A -85,B 0,C 180,E1 -30968.197,E2 -30968.197} C_VEL
LIN {X 0,Y 32.032,Z 578.742,A -85,B 0,C 180,E1 -30990.685,E2 -30990.685} C_VEL
LIN {X 0,Y 35.384,Z 581.167,A -85,B 0,C 180,E1 -30996.572,E2 -30996.572} C_VEL
LIN {X 0,Y 28.215,Z 575.254,A -85,B 0,C 180,E1 -31020.121,E2 -31020.121} C_VEL
LIN {X 0,Y 27.342,Z 573.583,A -85,B 0,C 180,E1 -31027.322,E2 -31027.322} C_VEL
LIN {X 0,Y 26.095,Z 570.447,A -85,B 0,C 180,E1 -31038.347,E2 -31038.347} C_VEL
LIN {X 0,Y 24.926,Z 565.093,A -85,B 0,C 180,E1 -31054.704,E2 -31054.704} C_VEL
LIN {X 0,Y 24.681,Z 561.251,A -85,B 0,C 180,E1 -31065.152,E2 -31065.152} C_VEL
LIN {X 0,Y 24.499,Z 557.107,A -85,B 0,C 180,E1 -31075.103,E2 -31075.103} C_VEL
LIN {X 0,Y 24.461,Z 554.226,A -85,B 0,C 180,E1 -31081.507,E2 -31081.507} C_VEL
LIN {X 0,Y 24.742,Z 548.191,A -85,B 0,C 180,E1 -31093.863,E2 -31093.863} C_VEL
LIN {X 0,Y 25.717,Z 541.911,A -85,B 0,C 180,E1 -31105.063,E2 -31105.063} C_VEL
LIN {X 0,Y 28.788,Z 530.179,A -85,B 0,C 180,E1 -31121.387,E2 -31121.387} C_VEL
LIN {X 0,Y 30.635,Z 523.731,A -85,B 0,C 180,E1 -31128.423,E2 -31128.423} C_VEL
LIN {X 0,Y 30.209,Z 519.09,A -85,B 0,C 180,E1 -31136.668,E2 -31136.668} C_VEL
LIN {X 0,Y 29.618,Z 513.112,A -85,B 0,C 180,E1 -31149.794,E2 -31149.794} C_VEL
LIN {X 0,Y 29.108,Z 511.788,A -85,B 0,C 180,E1 -31155.037,E2 -31155.037} C_VEL
LIN {X 0,Y 28.149,Z 509.879,A -85,B 0,C 180,E1 -31169.96,E2 -31169.96} C_VEL
LIN {X 0,Y 28.086,Z 509.729,A -85,B 0,C 180,E1 -31181.352,E2 -31181.352} C_VEL
LIN {X 0,Y 28.853,Z 512.277,A -85,B 0,C 180,E1 -31200.846,E2 -31200.846} C_VEL
LIN {X 0,Y 29.801,Z 514.889,A -85,B 0,C 180,E1 -31210.624,E2 -31210.624} C_VEL
LIN {X 0,Y 30.18,Z 519.324,A -85,B 0,C 180,E1 -31219.661,E2 -31219.661} C_VEL
LIN {X 0,Y 30.249,Z 526.475,A -85,B 0,C 180,E1 -31231.664,E2 -31231.664} C_VEL
LIN {X 0,Y 30.398,Z 530.561,A -85,B 0,C 180,E1 -31238.175,E2 -31238.175} C_VEL
LIN {X 0,Y 23.942,Z 540.777,A -85,B 0,C 180,E1 -31248.667,E2 -31248.667} C_VEL
LIN {X 0,Y 17.654,Z 551.935,A -85,B 0,C 180,E1 -31272.136,E2 -31272.136} C_VEL
LIN {X 0,Y 15.819,Z 560.971,A -85,B 0,C 180,E1 -31307.16,E2 -31307.16} C_VEL
LIN {X 0,Y 19.719,Z 569.069,A -85,B 0,C 180,E1 -31340.875,E2 -31340.875} C_VEL
LIN {X 0,Y 26.295,Z 575.056,A -85,B 0,C 180,E1 -31358.07,E2 -31358.07} C_VEL
LIN {X 0,Y 22.909,Z 572.157,A -85,B 0,C 180,E1 -31372.154,E2 -31372.154} C_VEL
LIN {X 0,Y 20.943,Z 569.349,A -85,B 0,C 180,E1 -31385.199,E2 -31385.199} C_VEL
LIN {X 0,Y 18.657,Z 564.402,A -85,B 0,C 180,E1 -31404.596,E2 -31404.596} C_VEL
LIN {X 0,Y 19.357,Z 555.342,A -85,B 0,C 180,E1 -31436.989,E2 -31436.989} C_VEL
LIN {X 0,Y 24.949,Z 544.556,A -85,B 0,C 180,E1 -31460.773,E2 -31460.773} C_VEL
LIN {X 0,Y 25.717,Z 541.911,A -85,B 0,C 180,E1 -31465.063,E2 -31465.063} C_VEL
LIN {X 0,Y 25.923,Z 538.824,A -85,B 0,C 180,E1 -31470.491,E2 -31470.491} C_VEL
LIN {X 0,Y 25.109,Z 533.965,A -85,B 0,C 180,E1 -31480.526,E2 -31480.526} C_VEL
LIN {X 0,Y 24.63,Z 528.042,A -85,B 0,C 180,E1 -31493.46,E2 -31493.46} C_VEL
LIN {X 0,Y 25.013,Z 525.879,A -85,B 0,C 180,E1 -31497.119,E2 -31497.119} C_VEL
LIN {X 0,Y 25.156,Z 524.415,A -85,B 0,C 180,E1 -31500.003,E2 -31500.003} C_VEL
LIN {X 0,Y 25.29,Z 519.66,A -85,B 0,C 180,E1 -31511.599,E2 -31511.599} C_VEL
LIN {X 0,Y 25.376,Z 518.067,A -85,B 0,C 180,E1 -31516.082,E2 -31516.082} C_VEL
LIN {X 0,Y 24.812,Z 516.166,A -85,B 0,C 180,E1 -31531.819,E2 -31531.819} C_VEL
LIN {X 0,Y 24.756,Z 516.114,A -85,B 0,C 180,E1 -31534.599,E2 -31534.599} C_VEL
LIN {X 0,Y 25.002,Z 518.035,A -85,B 0,C 180,E1 -31557.496,E2 -31557.496} C_VEL
LIN {X 0,Y 25.249,Z 520.459,A -85,B 0,C 180,E1 -31566.947,E2 -31566.947} C_VEL
LIN {X 0,Y 24.733,Z 525.269,A -85,B 0,C 180,E1 -31577.349,E2 -31577.349} C_VEL
LIN {X 0,Y 24.313,Z 530.698,A -85,B 0,C 180,E1 -31588.355,E2 -31588.355} C_VEL
LIN {X 0,Y 22.787,Z 533.271,A -85,B 0,C 180,E1 -31590.964,E2 -31590.964} C_VEL
LIN {X 0,Y 13.856,Z 545.585,A -85,B 0,C 180,E1 -31609.129,E2 -31609.129} C_VEL
LIN {X 0,Y 9.425,Z 553.986,A -85,B 0,C 180,E1 -31645.325,E2 -31645.325} C_VEL
LIN {X 0,Y 11.224,Z 561.977,A -85,B 0,C 180,E1 -31698.238,E2 -31698.238} C_VEL
LIN {X 0,Y 17.036,Z 567.799,A -85,B 0,C 180,E1 -31721.741,E2 -31721.741} C_VEL
LIN {X 0,Y 16.344,Z 566.999,A -85,B 0,C 180,E1 -31729.834,E2 -31729.834} C_VEL
LIN {X 0,Y 14.327,Z 564.591,A -85,B 0,C 180,E1 -31740.624,E2 -31740.624} C_VEL
LIN {X 0,Y 11.799,Z 555.909,A -85,B 0,C 180,E1 -31787.327,E2 -31787.327} C_VEL
LIN {X 0,Y 17.196,Z 545.513,A -85,B 0,C 180,E1 -31824.824,E2 -31824.824} C_VEL
LIN {X 0,Y 18.516,Z 543.584,A -85,B 0,C 180,E1 -31828.65,E2 -31828.65} C_VEL
LIN {X 0,Y 21.758,Z 534.4,A -85,B 0,C 180,E1 -31845.697,E2 -31845.697} C_VEL
LIN {X 0,Y 25.013,Z 525.879,A -85,B 0,C 180,E1 -31857.119,E2 -31857.119} C_VEL
LIN {X 0,Y 24.773,Z 524.763,A -85,B 0,C 180,E1 -31860.399,E2 -31860.399} C_VEL
LIN {X 0,Y 23.132,Z 524.318,A -85,B 0,C 180,E1 -31867.474,E2 -31867.474} C_VEL
LIN {X 0,Y 21.106,Z 524.275,A -85,B 0,C 180,E1 -31879.396,E2 -31879.396} C_VEL
LIN {X 0,Y 20.993,Z 523.846,A -85,B 0,C 180,E1 -31882.922,E2 -31882.922} C_VEL
LIN {X 0,Y 21.16,Z 522.887,A -85,B 0,C 180,E1 -31888.341,E2 -31888.341} C_VEL
LIN {X 0,Y 20.894,Z 523.017,A -85,B 0,C 180,E1 -31902.283,E2 -31902.283} C_VEL
LIN {X 0,Y 21.005,Z 524.088,A -85,B 0,C 180,E1 -31914.852,E2 -31914.852} C_VEL
LIN {X 0,Y 20.579,Z 525.805,A -85,B 0,C 180,E1 -31920.516,E2 -31920.516} C_VEL
LIN {X 0,Y 18.94,Z 531.633,A -85,B 0,C 180,E1 -31935.145,E2 -31935.145} C_VEL
LIN {X 0,Y 8.827,Z 543.985,A -85,B 0,C 180,E1 -31944.525,E2 -31944.525} C_VEL
LIN {X 0,Y 2.675,Z 553.585,A -85,B 0,C 180,E1 -32039.97,E2 -32039.97} C_VEL
LIN {X 0,Y 5.202,Z 556.812,A -85,B 0,C 180,E1 -32082.476,E2 -32082.476} C_VEL
LIN {X 0,Y 6.231,Z 557.404,A -85,B 0,C 180,E1 -32101.21,E2 -32101.21} C_VEL
LIN {X 0,Y 9.65,Z 546.184,A -85,B 0,C 180,E1 -32195.553,E2 -32195.553} C_VEL
LIN {X 0,Y 12.799,Z 542.426,A -85,B 0,C 180,E1 -32203.931,E2 -32203.931} C_VEL
LIN {X 0,Y 18.668,Z 530.827,A -85,B 0,C 180,E1 -32226.089,E2 -32226.089} C_VEL
LIN {X 0,Y 20.025,Z 528.178,A -85,B 0,C 180,E1 -32229.27,E2 -32229.27} C_VEL
LIN {X 0,Y 20.589,Z 526.181,A -85,B 0,C 180,E1 -32234.297,E2 -32234.297} C_VEL
LIN {X 0,Y 20.985,Z 524.435,A -85,B 0,C 180,E1 -32239.571,E2 -32239.571} C_VEL
LIN {X 0,Y 20.993,Z 523.846,A -85,B 0,C 180,E1 -32242.922,E2 -32242.922} C_VEL
LIN {X 0,Y 20.647,Z 523.844,A -85,B 0,C 180,E1 -32247.418,E2 -32247.418} C_VEL
LIN {X 0,Y 19.524,Z 525.289,A -85,B 0,C 180,E1 -32253.138,E2 -32253.138} C_VEL
LIN {X 0,Y 17.477,Z 528.431,A -85,B 0,C 180,E1 -32258.84,E2 -32258.84} C_VEL
LIN {X 0,Y 14.866,Z 532.449,A -85,B 0,C 180,E1 -32262.562,E2 -32262.562} C_VEL
LIN {X 0,Y 11.88,Z 536.744,A -85,B 0,C 180,E1 -32264.487,E2 -32264.487} C_VEL
LIN {X 0,Y 8.754,Z 540.79,A -85,B 0,C 180,E1 -32260.247,E2 -32260.247} C_VEL
LIN {X 0,Y 7.752,Z 542.104,A -85,B 0,C 180,E1 -32256.263,E2 -32256.263} C_VEL
LIN {X 0,Y 7.405,Z 543.097,A -85,B 0,C 180,E1 -32238.376,E2 -32238.376} C_VEL
LIN {X 0,Y 8.43,Z 541.952,A -85,B 0,C 180,E1 -32236.916,E2 -32236.916} C_VEL
LIN {X 0,Y 13.304,Z 535.099,A -85,B 0,C 180,E1 -32244.642,E2 -32244.642} C_VEL
LIN {X 0,Y 15.91,Z 531.183,A -85,B 0,C 180,E1 -32247.936,E2 -32247.936} C_VEL
LIN {X 0,Y 16.985,Z 529.371,A -85,B 0,C 180,E1 -32250.489,E2 -32250.489} C_VEL
LIN {X 0,Y 17.133,Z 528.971,A -85,B 0,C 180,E1 -32254.875,E2 -32254.875} C_VEL
LIN {X 0,Y 17.024,Z 529.313,A -85,B 0,C 180,E1 -32264.742,E2 -32264.742} C_VEL
LIN {X 0,Y 15.878,Z 531.418,A -85,B 0,C 180,E1 -32270.366,E2 -32270.366} C_VEL
LIN {X 0,Y 14.694,Z 533.176,A -85,B 0,C 180,E1 -32271.653,E2 -32271.653} C_VEL
LIN {X 0,Y 8.754,Z 540.79,A -85,B 0,C 180,E1 -32260.247,E2 -32260.247} C_VEL
LIN {X 0,Y 8.317,Z 542.11,A -85,B 0,C 180,E1 -32258.648,E2 -32258.648} C_VEL
LIN {X 0,Y 8.317,Z 600,A -85,B 0,C 180,E1 -32258.648,E2 -32258.648} C_VEL
LIN {X 0,Y 8.317,Z 600,A -85,B 0,C 180,E1 -32258.648,E2 -32258.648}

QRS_NEXT_CUT()

QRS_NEXT()
QRS_HOME()

END
